C05496=1168.158,-99.130,-41.882,178.959,5.803,149.342
C05497=1168.163,-99.379,-41.873,178.956,5.803,149.343
C05498=1168.169,-99.629,-41.863,178.955,5.803,149.343
C05499=1168.174,-99.879,-41.854,178.952,5.803,149.344
C05500=1168.180,-100.128,-41.844,178.950,5.803,149.344
C05501=1168.185,-100.378,-41.835,178.948,5.802,149.345
C05502=1168.189,-100.629,-41.825,178.946,5.801,149.346
C05503=1168.195,-100.878,-41.815,178.944,5.802,149.346
C05504=1168.200,-101.128,-41.806,178.941,5.801,149.347
C05505=1168.206,-101.378,-41.796,178.940,5.801,149.347
C05506=1168.211,-101.628,-41.787,178.937,5.801,149.348
C05507=1168.216,-101.900,-41.777,178.935,5.800,149.349
C05508=1168.223,-102.171,-41.767,178.933,5.800,149.349
C05509=1168.229,-102.443,-41.756,178.930,5.800,149.350
C05510=1168.234,-102.715,-41.746,178.928,5.799,149.350
C05511=1168.239,-102.965,-41.737,178.926,5.799,149.351
C05512=1168.245,-103.214,-41.727,178.924,5.799,149.352
C05513=1168.250,-103.464,-41.718,178.922,5.799,149.352
C05514=1168.255,-103.714,-41.709,178.919,5.799,149.353
C05515=1168.261,-103.964,-41.699,178.917,5.798,149.353
C05516=1168.266,-104.213,-41.690,178.915,5.798,149.354
C05517=1168.271,-104.463,-41.681,178.913,5.797,149.355
C05518=1168.277,-104.713,-41.671,178.911,5.797,149.355
C05519=1168.282,-104.963,-41.662,178.909,5.797,149.356
C05520=1168.288,-105.213,-41.653,178.907,5.797,149.356
C05521=1168.293,-105.462,-41.643,178.905,5.796,149.357
C05522=1168.298,-105.712,-41.634,178.902,5.796,149.357
C05523=1168.304,-105.962,-41.625,178.900,5.796,149.358
C05524=1168.309,-106.211,-41.615,178.898,5.795,149.358
C05525=1168.314,-106.461,-41.606,178.896,5.796,149.359
C05526=1168.319,-106.711,-41.597,178.894,5.795,149.360
C05527=1168.325,-106.961,-41.588,178.892,5.795,149.360
C05528=1168.330,-107.210,-41.578,178.890,5.795,149.361
C05529=1168.335,-107.460,-41.569,178.888,5.795,149.361
C05530=1168.341,-107.710,-41.560,178.885,5.794,149.362
C05531=1168.346,-107.960,-41.551,178.883,5.793,149.362
C05532=1168.351,-108.209,-41.541,178.881,5.794,149.363
C05533=1168.357,-108.460,-41.532,178.879,5.793,149.364
C05534=1168.362,-108.709,-41.523,178.877,5.793,149.364
C05535=1168.367,-108.959,-41.514,178.875,5.793,149.365
C05536=1168.372,-109.209,-41.505,178.873,5.793,149.365
C05537=1168.378,-109.459,-41.495,178.871,5.792,149.366
C05538=1168.383,-109.709,-41.486,178.869,5.792,149.367
C05539=1168.388,-109.958,-41.477,178.867,5.792,149.367
C05540=1168.393,-110.208,-41.468,178.865,5.792,149.368
C05541=1168.400,-110.458,-41.459,178.862,5.791,149.368
C05542=1168.405,-110.707,-41.449,178.860,5.790,149.369
C05543=1168.410,-110.957,-41.440,178.858,5.791,149.369
C05544=1168.415,-111.207,-41.432,178.856,5.790,149.370
C05545=1168.421,-111.457,-41.422,178.854,5.790,149.370
C05546=1168.426,-111.707,-41.413,178.852,5.790,149.371
C05547=1168.431,-111.957,-41.404,178.850,5.790,149.372
C05548=1168.437,-112.206,-41.395,178.848,5.789,149.372
C05549=1168.442,-112.456,-41.386,178.846,5.789,149.373
C05550=1168.447,-112.706,-41.376,178.844,5.789,149.373
C05551=1168.452,-112.956,-41.367,178.842,5.789,149.374
C05552=1168.458,-113.206,-41.358,178.839,5.788,149.375
C05553=1168.463,-113.455,-41.350,178.838,5.788,149.375
C05554=1168.469,-113.704,-41.341,178.835,5.788,149.376
C05555=1168.474,-113.955,-41.331,178.833,5.787,149.376
C05556=1168.480,-114.205,-41.323,178.831,5.787,149.377
C05557=1168.485,-114.454,-41.314,178.829,5.787,149.377
C05558=1168.490,-114.704,-41.305,178.827,5.787,149.378
C05559=1168.495,-114.954,-41.296,178.825,5.786,149.378
C05560=1168.500,-115.204,-41.287,178.823,5.787,149.379
C05561=1168.507,-115.453,-41.278,178.820,5.786,149.380
C05562=1168.512,-115.703,-41.269,178.819,5.786,149.380
C05563=1168.517,-115.953,-41.260,178.816,5.785,149.381
C05564=1168.522,-116.203,-41.251,178.815,5.785,149.381
C05565=1168.528,-116.453,-41.242,178.812,5.785,149.382
C05566=1168.533,-116.703,-41.233,178.810,5.785,149.382
C05567=1168.538,-116.952,-41.224,178.808,5.784,149.383
C05568=1168.544,-117.202,-41.215,178.807,5.784,149.383
C05569=1168.550,-117.452,-41.206,178.804,5.784,149.384
C05570=1168.555,-117.702,-41.198,178.802,5.784,149.385
C05571=1168.560,-117.952,-41.189,178.800,5.783,149.385
C05572=1168.565,-118.201,-41.180,178.798,5.784,149.386
C05573=1168.570,-118.451,-41.171,178.796,5.783,149.386
C05574=1168.576,-118.700,-41.162,178.794,5.783,149.387
C05575=1168.581,-118.950,-41.153,178.792,5.783,149.388
C05576=1168.586,-119.200,-41.145,178.790,5.783,149.388
C05577=1168.591,-119.450,-41.136,178.788,5.782,149.389
C05578=1168.597,-119.700,-41.127,178.785,5.782,149.389
C05579=1168.603,-119.950,-41.117,178.783,5.782,149.390
C05580=1168.608,-120.199,-41.109,178.781,5.781,149.390
C05581=1168.613,-120.449,-41.100,178.779,5.781,149.391
C05582=1168.619,-120.699,-41.091,178.777,5.780,149.391
C05583=1168.624,-120.949,-41.082,178.775,5.780,149.392
C05584=1168.629,-121.198,-41.073,178.773,5.780,149.392
C05585=1168.635,-121.448,-41.065,178.771,5.780,149.393
C05586=1168.640,-121.698,-41.056,178.769,5.779,149.394
C05587=1168.645,-121.948,-41.048,178.767,5.779,149.394
C05588=1168.651,-122.198,-41.039,178.765,5.779,149.395
C05589=1168.656,-122.448,-41.030,178.763,5.779,149.395
C05590=1168.661,-122.697,-41.021,178.761,5.778,149.396
C05591=1168.667,-122.947,-41.012,178.759,5.779,149.396
C05592=1168.672,-123.197,-41.003,178.757,5.778,149.397
C05593=1168.677,-123.447,-40.995,178.755,5.778,149.397
C05594=1168.683,-123.696,-40.987,178.752,5.778,149.398
C05595=1168.688,-123.946,-40.978,178.751,5.778,149.399
C05596=1168.693,-124.196,-40.969,178.748,5.777,149.399
C05597=1168.699,-124.446,-40.960,178.747,5.777,149.400
C05598=1168.705,-124.695,-40.952,178.744,5.777,149.400
C05599=1168.710,-124.945,-40.943,178.743,5.777,149.401
C05600=1168.715,-125.195,-40.934,178.740,5.776,149.401
C05601=1168.720,-125.445,-40.925,178.738,5.776,149.402
C05602=1168.726,-125.694,-40.917,178.736,5.775,149.403
C05603=1168.731,-125.945,-40.909,178.735,5.776,149.403
C05604=1168.736,-126.194,-40.900,178.732,5.775,149.403
C05605=1168.742,-126.444,-40.891,178.730,5.775,149.404
C05606=1168.747,-126.693,-40.882,178.729,5.775,149.405
C05607=1168.753,-126.944,-40.874,178.726,5.774,149.405
C05608=1168.757,-127.193,-40.866,178.724,5.775,149.406
C05609=1168.762,-127.443,-40.857,178.722,5.774,149.406
C05610=1168.768,-127.692,-40.849,178.721,5.774,149.407
C05611=1168.347,-127.704,-40.890,178.717,5.777,149.409
C05612=1168.342,-127.455,-40.898,178.718,5.777,149.408
C05613=1168.337,-127.205,-40.907,178.720,5.778,149.408
C05614=1168.331,-126.954,-40.915,178.723,5.778,149.407
C05615=1168.326,-126.704,-40.924,178.725,5.778,149.407
C05616=1168.320,-126.455,-40.933,178.726,5.778,149.406
C05617=1168.315,-126.205,-40.942,178.729,5.779,149.405
C05618=1168.309,-125.955,-40.950,178.731,5.779,149.405
C05619=1168.304,-125.706,-40.958,178.733,5.780,149.404
C05620=1168.299,-125.456,-40.967,178.734,5.779,149.404
C05621=1168.294,-125.206,-40.976,178.737,5.780,149.403
C05622=1168.289,-124.956,-40.984,178.739,5.780,149.403
C05623=1168.283,-124.707,-40.992,178.741,5.781,149.402
C05624=1168.278,-124.457,-41.001,178.743,5.780,149.401
C05625=1168.273,-124.207,-41.010,178.745,5.781,149.401
C05626=1168.267,-123.957,-41.019,178.747,5.781,149.400
C05627=1168.262,-123.708,-41.027,178.749,5.782,149.400
C05628=1168.256,-123.458,-41.036,178.751,5.781,149.399
C05629=1168.251,-123.208,-41.045,178.753,5.782,149.399
C05630=1168.246,-122.958,-41.053,178.755,5.782,149.398
C05631=1168.241,-122.708,-41.062,178.758,5.782,149.398
C05632=1168.235,-122.459,-41.071,178.759,5.782,149.397
C05633=1168.230,-122.209,-41.080,178.761,5.783,149.397
C05634=1168.224,-121.959,-41.088,178.763,5.783,149.396
C05635=1168.219,-121.709,-41.097,178.766,5.783,149.395
C05636=1168.213,-121.460,-41.105,178.767,5.783,149.395
C05637=1168.208,-121.210,-41.114,178.769,5.784,149.394
C05638=1168.203,-120.960,-41.123,178.771,5.784,149.394
C05639=1168.197,-120.710,-41.133,178.774,5.784,149.393
C05640=1168.192,-120.460,-41.142,178.775,5.784,149.393
C05641=1168.186,-120.211,-41.150,178.778,5.785,149.392
C05642=1168.181,-119.961,-41.159,178.780,5.785,149.392
C05643=1168.176,-119.711,-41.168,178.782,5.786,149.391
C05644=1168.170,-119.460,-41.176,178.784,5.785,149.390
C05645=1168.165,-119.211,-41.185,178.786,5.786,149.390
C05646=1168.160,-118.961,-41.194,178.788,5.786,149.389
C05647=1168.154,-118.712,-41.202,178.790,5.786,149.389
C05648=1168.149,-118.462,-41.211,178.792,5.786,149.388
C05649=1168.144,-118.212,-41.220,178.794,5.787,149.388
C05650=1168.139,-117.962,-41.229,178.796,5.787,149.387
C05651=1168.134,-117.712,-41.238,178.798,5.787,149.386
C05652=1168.128,-117.462,-41.247,178.800,5.787,149.386
C05653=1168.122,-117.213,-41.256,178.803,5.788,149.385
C05654=1168.117,-116.963,-41.265,178.804,5.788,149.385
C05655=1168.112,-116.713,-41.274,178.806,5.788,149.384
C05656=1168.106,-116.463,-41.283,178.809,5.788,149.384
C05657=1168.101,-116.214,-41.292,178.811,5.789,149.383
C05658=1168.096,-115.964,-41.301,178.813,5.789,149.383
C05659=1168.090,-115.715,-41.309,178.815,5.789,149.382
C05660=1168.084,-115.464,-41.319,178.817,5.790,149.381
C05661=1168.079,-115.214,-41.327,178.819,5.790,149.381
C05662=1168.074,-114.965,-41.336,178.821,5.790,149.380
C05663=1168.069,-114.715,-41.345,178.823,5.790,149.380
C05664=1168.064,-114.465,-41.354,178.825,5.791,149.379
C05665=1168.059,-114.215,-41.363,178.827,5.790,149.379
C05666=1168.053,-113.965,-41.373,178.830,5.791,149.378
C05667=1168.047,-113.716,-41.382,178.831,5.791,149.378
C05668=1168.042,-113.467,-41.391,178.834,5.792,149.377
C05669=1168.037,-113.217,-41.400,178.835,5.792,149.376
C05670=1168.032,-112.967,-41.408,178.838,5.792,149.376
C05671=1168.027,-112.717,-41.417,178.840,5.792,149.375
C05672=1168.021,-112.467,-41.427,178.842,5.793,149.375
C05673=1168.015,-112.217,-41.436,178.843,5.793,149.374
C05674=1168.010,-111.967,-41.445,178.846,5.793,149.373
C05675=1168.005,-111.717,-41.454,178.848,5.794,149.373
C05676=1168.000,-111.468,-41.464,178.850,5.794,149.372
C05677=1167.994,-111.219,-41.472,178.853,5.794,149.372
C05678=1167.989,-110.969,-41.481,178.854,5.794,149.371
C05679=1167.983,-110.719,-41.490,178.857,5.794,149.371
C05680=1167.978,-110.469,-41.499,178.858,5.794,149.370
C05681=1167.972,-110.219,-41.508,178.861,5.795,149.370
C05682=1167.967,-109.969,-41.517,178.863,5.795,149.369
C05683=1167.962,-109.720,-41.527,178.865,5.796,149.368
C05684=1167.957,-109.470,-41.536,178.867,5.796,149.368
C05685=1167.951,-109.220,-41.545,178.869,5.796,149.367
C05686=1167.946,-108.970,-41.554,178.871,5.797,149.367
C05687=1167.941,-108.720,-41.563,178.873,5.797,149.366
C05688=1167.935,-108.471,-41.573,178.876,5.797,149.366
C05689=1167.930,-108.221,-41.582,178.877,5.797,149.365
C05690=1167.925,-107.971,-41.591,178.880,5.797,149.364
C05691=1167.920,-107.721,-41.600,178.882,5.797,149.364
C05692=1167.914,-107.471,-41.610,178.884,5.798,149.363
C05693=1167.909,-107.222,-41.619,178.886,5.798,149.363
C05694=1167.904,-106.972,-41.628,178.888,5.798,149.362
C05695=1167.898,-106.722,-41.638,178.890,5.799,149.362
C05696=1167.893,-106.472,-41.647,178.892,5.799,149.361
C05697=1167.888,-106.222,-41.656,178.895,5.800,149.360
C05698=1167.883,-105.973,-41.665,178.897,5.799,149.360
C05699=1167.877,-105.722,-41.674,178.899,5.800,149.359
C05700=1167.872,-105.473,-41.684,178.900,5.800,149.359
C05701=1167.867,-105.223,-41.693,178.903,5.800,149.358
C05702=1167.861,-104.973,-41.702,178.905,5.800,149.358
C05703=1167.856,-104.724,-41.712,178.907,5.801,149.357
C05704=1167.851,-104.474,-41.721,178.910,5.801,149.356
C05705=1167.845,-104.224,-41.730,178.911,5.801,149.356
C05706=1167.840,-103.975,-41.740,178.914,5.802,149.355
C05707=1167.834,-103.725,-41.750,178.915,5.802,149.355
C05708=1167.829,-103.475,-41.758,178.918,5.803,149.354
C05709=1167.824,-103.226,-41.768,178.920,5.802,149.354
C05710=1167.818,-102.975,-41.778,178.922,5.803,149.353
C05711=1167.813,-102.725,-41.786,178.925,5.803,149.352
C05712=1167.807,-102.454,-41.796,178.926,5.803,149.352
C05713=1167.802,-102.182,-41.807,178.929,5.804,149.351
C05714=1167.795,-101.910,-41.817,178.931,5.804,149.351
C05715=1167.790,-101.638,-41.828,178.933,5.804,149.350
C05716=1167.785,-101.389,-41.837,178.936,5.804,149.349
C05717=1167.779,-101.139,-41.847,178.938,5.805,149.349
C05718=1167.774,-100.889,-41.856,178.940,5.805,149.348
C05719=1167.769,-100.640,-41.865,178.942,5.805,149.348
C05720=1167.763,-100.390,-41.875,178.944,5.805,149.347
C05721=1167.758,-100.140,-41.884,178.947,5.806,149.346
C05722=1167.752,-99.890,-41.894,178.948,5.806,149.346
C05723=1167.748,-99.641,-41.903,178.950,5.807,149.345
C05724=1167.742,-99.391,-41.913,178.953,5.807,149.345
C05725=1167.736,-99.141,-41.922,178.955,5.807,149.344
C05726=1167.731,-98.891,-41.932,178.957,5.807,149.343
C05727=1167.726,-98.641,-41.941,178.959,5.807,149.343
C05728=1167.721,-98.391,-41.952,178.961,5.808,149.342
C05729=1167.716,-98.141,-41.960,178.964,5.808,149.342
C05730=1167.710,-97.892,-41.971,178.965,5.808,149.341
C05731=1167.705,-97.642,-41.980,178.968,5.809,149.341
C05732=1167.700,-97.393,-41.989,178.970,5.809,149.340
C05733=1167.694,-97.143,-41.999,178.972,5.810,149.340
C05734=1167.689,-96.893,-42.008,178.974,5.810,149.339
C05735=1167.683,-96.643,-42.018,178.976,5.810,149.338
C05736=1167.678,-96.394,-42.028,178.979,5.810,149.338
C05737=1167.673,-96.143,-42.037,178.980,5.810,149.337
C05738=1167.667,-95.894,-42.047,178.983,5.811,149.336
C05739=1167.663,-95.644,-42.057,178.985,5.811,149.336
C05740=1167.657,-95.394,-42.067,178.987,5.811,149.336
C05741=1167.652,-95.145,-42.076,178.989,5.812,149.335
C05742=1167.646,-94.895,-42.086,178.991,5.812,149.334
C05743=1167.641,-94.646,-42.095,178.994,5.812,149.334
C05744=1167.635,-94.395,-42.105,178.996,5.813,149.333
C05745=1167.631,-94.145,-42.115,178.998,5.813,149.332
C05746=1167.625,-93.896,-42.125,179.000,5.813,149.332
C05747=1167.620,-93.646,-42.134,179.002,5.813,149.331
C05748=1167.615,-93.397,-42.144,179.004,5.814,149.331
C05749=1167.609,-93.146,-42.154,179.007,5.815,149.330
C05750=1167.604,-92.897,-42.163,179.009,5.814,149.330
C05751=1167.599,-92.647,-42.174,179.011,5.815,149.329
C05752=1167.594,-92.397,-42.183,179.013,5.814,149.328
C05753=1167.588,-92.148,-42.193,179.015,5.815,149.328
C05754=1167.583,-91.898,-42.202,179.018,5.816,149.327
C05755=1167.577,-91.648,-42.212,179.019,5.816,149.327
C05756=1167.572,-91.399,-42.222,179.022,5.816,149.326
C05757=1167.567,-91.149,-42.232,179.024,5.816,149.325
C05758=1167.561,-90.898,-42.242,179.026,5.817,149.325
C05759=1167.556,-90.649,-42.252,179.029,5.817,149.324
C05760=1167.551,-90.400,-42.261,179.030,5.817,149.324
C05761=1167.545,-90.150,-42.271,179.033,5.818,149.323
C05762=1167.541,-89.900,-42.281,179.035,5.818,149.323
C05763=1167.535,-89.650,-42.291,179.037,5.818,149.322
C05764=1167.529,-89.400,-42.301,179.039,5.819,149.321
C05765=1167.525,-89.151,-42.310,179.041,5.819,149.321
C05766=1167.519,-88.901,-42.320,179.044,5.819,149.320
C05767=1167.514,-88.651,-42.331,179.046,5.820,149.320
C05768=1167.509,-88.401,-42.340,179.048,5.819,149.319
C05769=1167.503,-88.151,-42.350,179.050,5.820,149.319
C05770=1167.498,-87.902,-42.360,179.053,5.821,149.318
C05771=1167.493,-87.653,-42.370,179.054,5.821,149.317
C05772=1167.487,-87.402,-42.380,179.057,5.821,149.317
C05773=1167.482,-87.152,-42.390,179.059,5.821,149.316
C05774=1167.477,-86.903,-42.400,179.061,5.821,149.315
C05775=1167.471,-86.654,-42.410,179.063,5.822,149.315
C05776=1167.466,-86.403,-42.420,179.065,5.822,149.314
C05777=1167.461,-86.153,-42.429,179.068,5.822,149.314
C05778=1167.456,-85.904,-42.440,179.070,5.823,149.313
C05779=1167.450,-85.654,-42.450,179.072,5.823,149.313
C05780=1167.445,-85.404,-42.460,179.074,5.824,149.312
C05781=1167.440,-85.155,-42.470,179.077,5.824,149.311
C05782=1167.435,-84.905,-42.480,179.078,5.824,149.311
C05783=1167.429,-84.654,-42.490,179.081,5.824,149.310
C05784=1167.424,-84.405,-42.500,179.083,5.825,149.310
C05785=1167.419,-84.156,-42.510,179.085,5.825,149.309
C05786=1167.413,-83.906,-42.520,179.088,5.826,149.309
C05787=1167.408,-83.656,-42.531,179.090,5.825,149.308
C05788=1167.403,-83.407,-42.540,179.092,5.826,149.307
C05789=1167.398,-83.157,-42.550,179.094,5.827,149.307
C05790=1167.393,-82.907,-42.561,179.096,5.826,149.306
C05791=1167.387,-82.657,-42.571,179.098,5.827,149.306
C05792=1167.382,-82.407,-42.580,179.101,5.827,149.305
C05793=1167.376,-82.158,-42.590,179.103,5.827,149.304
C05794=1167.371,-81.908,-42.601,179.105,5.828,149.304
C05795=1167.366,-81.658,-42.611,179.107,5.829,149.303
C05796=1167.360,-81.409,-42.621,179.110,5.828,149.303
C05797=1167.356,-81.159,-42.631,179.112,5.829,149.302
C05798=1167.350,-80.909,-42.641,179.114,5.829,149.301
C05799=1167.345,-80.660,-42.652,179.116,5.829,149.301
C05800=1167.340,-80.409,-42.662,179.119,5.830,149.300
C05801=1167.334,-80.160,-42.672,179.121,5.831,149.300
C05802=1167.328,-79.910,-42.683,179.123,5.830,149.299
C05803=1167.324,-79.660,-42.693,179.125,5.831,149.299
C05804=1167.319,-79.411,-42.703,179.128,5.831,149.298
C05805=1167.313,-79.161,-42.713,179.129,5.831,149.297
C05806=1167.308,-78.911,-42.724,179.132,5.832,149.297
C05807=1167.302,-78.661,-42.734,179.134,5.833,149.296
C05808=1167.297,-78.412,-42.744,179.136,5.832,149.295
C05809=1167.292,-78.162,-42.755,179.138,5.833,149.295
C05810=1167.287,-77.912,-42.764,179.141,5.833,149.294
C05811=1167.281,-77.663,-42.774,179.143,5.833,149.294
C05812=1167.276,-77.413,-42.785,179.145,5.834,149.293
C05813=1167.271,-77.163,-42.795,179.148,5.834,149.293
C05814=1167.265,-76.914,-42.805,179.150,5.834,149.292
C05815=1167.260,-76.663,-42.816,179.152,5.835,149.291
C05816=1167.254,-76.393,-42.827,179.155,5.835,149.291
C05817=1167.249,-76.122,-42.839,179.157,5.836,149.290
C05818=1167.243,-75.850,-42.850,179.159,5.836,149.289
C05819=1167.237,-75.580,-42.861,179.162,5.836,149.289
C05820=1167.232,-75.329,-42.872,179.164,5.837,149.288
C05821=1167.226,-75.080,-42.882,179.166,5.837,149.288
C05822=1167.221,-74.829,-42.892,179.168,5.837,149.287
C05823=1167.216,-74.580,-42.903,179.171,5.838,149.286
C05824=1167.211,-74.331,-42.913,179.173,5.838,149.286
C05825=1167.206,-74.081,-42.924,179.175,5.838,149.285
C05826=1167.200,-73.831,-42.934,179.177,5.839,149.285
C05827=1167.195,-73.581,-42.945,179.180,5.839,149.284
C05828=1167.189,-73.331,-42.955,179.182,5.840,149.284
C05829=1167.184,-73.081,-42.966,179.184,5.840,149.283
C05830=1167.179,-72.832,-42.976,179.186,5.840,149.282
C05831=1167.174,-72.583,-42.987,179.189,5.841,149.282
C05832=1167.169,-72.332,-42.997,179.190,5.841,149.281
C05833=1167.163,-72.083,-43.007,179.193,5.841,149.280
C05834=1167.158,-71.833,-43.018,179.195,5.842,149.280
C05835=1167.152,-71.583,-43.028,179.197,5.842,149.279
C05836=1167.148,-71.334,-43.040,179.200,5.842,149.279
C05837=1167.142,-71.084,-43.050,179.202,5.843,149.278
C05838=1167.136,-70.834,-43.060,179.204,5.844,149.278
C05839=1167.131,-70.584,-43.071,179.207,5.843,149.277
C05840=1167.126,-70.335,-43.081,179.209,5.844,149.276
C05841=1167.121,-70.085,-43.092,179.211,5.844,149.276
C05842=1167.116,-69.835,-43.102,179.213,5.844,149.275
C05843=1167.111,-69.585,-43.113,179.216,5.845,149.274
C05844=1167.105,-69.336,-43.124,179.218,5.845,149.274
C05845=1167.100,-69.086,-43.134,179.220,5.845,149.273
C05846=1167.095,-68.837,-43.145,179.222,5.846,149.273
C05847=1167.090,-68.587,-43.156,179.225,5.846,149.272
C05848=1167.084,-68.337,-43.166,179.227,5.847,149.271
C05849=1167.079,-68.087,-43.177,179.229,5.847,149.271
C05850=1167.074,-67.838,-43.188,179.232,5.847,149.270
C05851=1167.069,-67.588,-43.198,179.234,5.848,149.270
C05852=1167.063,-67.338,-43.209,179.236,5.847,149.269
C05853=1167.058,-67.088,-43.220,179.238,5.848,149.269
C05854=1167.052,-66.839,-43.230,179.241,5.849,149.268
C05855=1167.047,-66.589,-43.241,179.243,5.849,149.267
C05856=1167.042,-66.340,-43.252,179.245,5.849,149.267
C05857=1167.037,-66.090,-43.263,179.247,5.850,149.266
C05858=1167.032,-65.840,-43.273,179.250,5.850,149.265
C05859=1167.027,-65.590,-43.284,179.252,5.851,149.265
C05860=1167.021,-65.341,-43.294,179.254,5.851,149.264
C05861=1167.016,-65.091,-43.306,179.256,5.851,149.264
C05862=1167.010,-64.841,-43.316,179.259,5.852,149.263
C05863=1167.005,-64.591,-43.327,179.261,5.852,149.263
C05864=1167.001,-64.341,-43.338,179.263,5.852,149.262
C05865=1166.995,-64.092,-43.348,179.266,5.853,149.261
C05866=1166.990,-63.842,-43.360,179.268,5.853,149.261
C05867=1166.985,-63.593,-43.370,179.270,5.853,149.260
C05868=1166.979,-63.343,-43.382,179.272,5.854,149.260
C05869=1166.974,-63.093,-43.392,179.275,5.855,149.259
C05870=1166.969,-62.844,-43.403,179.277,5.855,149.258
C05871=1166.963,-62.594,-43.413,179.279,5.855,149.258
C05872=1166.958,-62.344,-43.424,179.282,5.855,149.257
C05873=1166.953,-62.094,-43.436,179.284,5.856,149.256
C05874=1166.947,-61.844,-43.446,179.286,5.857,149.256
C05875=1166.943,-61.595,-43.457,179.289,5.856,149.255
C05876=1166.937,-61.345,-43.468,179.291,5.857,149.255
C05877=1166.932,-61.096,-43.479,179.293,5.857,149.254
C05878=1166.927,-60.846,-43.491,179.296,5.858,149.254
C05879=1166.921,-60.596,-43.501,179.298,5.858,149.253
C05880=1166.917,-60.346,-43.512,179.300,5.859,149.252
C05881=1166.911,-60.097,-43.523,179.302,5.859,149.252
C05882=1166.906,-59.847,-43.534,179.305,5.860,149.251
C05883=1166.901,-59.597,-43.545,179.307,5.859,149.251
C05884=1166.895,-59.348,-43.556,179.309,5.860,149.250
C05885=1166.890,-59.098,-43.566,179.312,5.861,149.249
C05886=1166.886,-58.848,-43.578,179.314,5.861,149.249
C05887=1166.880,-58.599,-43.589,179.316,5.861,149.248
C05888=1166.875,-58.348,-43.600,179.319,5.861,149.247
C05889=1166.869,-58.100,-43.611,179.321,5.862,149.247
C05890=1166.864,-57.849,-43.622,179.323,5.863,149.246
C05891=1166.859,-57.599,-43.633,179.325,5.863,149.246
C05892=1166.854,-57.350,-43.644,179.328,5.863,149.245
C05893=1166.849,-57.100,-43.655,179.330,5.864,149.245
C05894=1166.843,-56.850,-43.667,179.332,5.864,149.244
C05895=1166.838,-56.601,-43.678,179.334,5.864,149.243
C05896=1166.833,-56.351,-43.688,179.337,5.865,149.243
C05897=1166.827,-56.101,-43.700,179.339,5.865,149.242
C05898=1166.822,-55.852,-43.711,179.342,5.866,149.242
C05899=1166.817,-55.602,-43.722,179.344,5.866,149.241
C05900=1166.812,-55.352,-43.733,179.346,5.866,149.240
C05901=1166.806,-55.103,-43.744,179.349,5.867,149.240
C05902=1166.801,-54.853,-43.755,179.351,5.868,149.239
C05903=1166.796,-54.603,-43.767,179.353,5.868,149.239
C05904=1166.791,-54.354,-43.778,179.355,5.868,149.238
C05905=1166.786,-54.104,-43.789,179.358,5.868,149.237
C05906=1166.780,-53.854,-43.800,179.360,5.869,149.237
C05907=1166.776,-53.604,-43.811,179.363,5.870,149.236
C05908=1166.770,-53.355,-43.822,179.365,5.870,149.235
C05909=1166.765,-53.105,-43.834,179.367,5.870,149.235
C05910=1166.760,-52.855,-43.845,179.369,5.870,149.234
C05911=1166.754,-52.606,-43.856,179.372,5.871,149.234
C05912=1166.749,-52.356,-43.868,179.374,5.872,149.233
C05913=1166.744,-52.107,-43.879,179.376,5.872,149.233
C05914=1166.739,-51.856,-43.890,179.379,5.872,149.232
C05915=1166.733,-51.607,-43.901,179.381,5.873,149.231
C05916=1166.728,-51.357,-43.913,179.383,5.873,149.231
C05917=1166.723,-51.108,-43.924,179.386,5.874,149.230
C05918=1166.719,-50.858,-43.935,179.388,5.874,149.230
C05919=1166.712,-50.608,-43.946,179.390,5.874,149.229
C05920=1166.707,-50.338,-43.959,179.392,5.875,149.228
C05921=1166.701,-50.067,-43.972,179.395,5.875,149.228
C05922=1166.695,-49.797,-43.984,179.398,5.876,149.227
C05923=1166.691,-49.526,-43.996,179.401,5.876,149.226
C05924=1166.685,-49.277,-44.008,179.403,5.877,149.226
C05925=1166.680,-49.028,-44.019,179.405,5.877,149.225
C05926=1166.674,-48.777,-44.030,179.407,5.877,149.225
C05927=1166.669,-48.527,-44.041,179.410,5.878,149.224
C05928=1166.664,-48.277,-44.053,179.412,5.878,149.223
C05929=1166.659,-48.029,-44.064,179.414,5.879,149.223
C05930=1166.653,-47.779,-44.076,179.417,5.879,149.222
C05931=1166.649,-47.529,-44.087,179.419,5.880,149.222
C05932=1166.643,-47.279,-44.099,179.421,5.880,149.221
C05933=1166.638,-47.029,-44.110,179.424,5.881,149.220
C05934=1166.632,-46.780,-44.122,179.426,5.881,149.220
C05935=1166.627,-46.530,-44.134,179.428,5.882,149.219
C05936=1166.622,-46.281,-44.145,179.431,5.882,149.218
C05937=1166.617,-46.031,-44.157,179.433,5.882,149.218
C05938=1166.612,-45.781,-44.168,179.435,5.883,149.217
C05939=1166.606,-45.532,-44.180,179.438,5.883,149.217
C05940=1166.601,-45.282,-44.191,179.440,5.884,149.216
C05941=1166.596,-45.032,-44.203,179.443,5.884,149.215
C05942=1166.591,-44.783,-44.214,179.445,5.885,149.215
C05943=1166.586,-44.533,-44.226,179.447,5.885,149.214
C05944=1166.581,-44.284,-44.237,179.450,5.885,149.214
C05945=1166.575,-44.034,-44.249,179.452,5.886,149.213
C05946=1166.570,-43.784,-44.261,179.455,5.886,149.212
C05947=1166.565,-43.534,-44.272,179.457,5.887,149.212
C05948=1166.560,-43.284,-44.284,179.459,5.887,149.211
C05949=1166.555,-43.035,-44.295,179.461,5.888,149.211
C05950=1166.550,-42.785,-44.307,179.464,5.888,149.210
C05951=1166.543,-42.536,-44.319,179.466,5.889,149.210
C05952=1166.539,-42.286,-44.330,179.469,5.889,149.209
C05953=1166.533,-42.036,-44.342,179.471,5.890,149.208
C05954=1166.528,-41.786,-44.354,179.473,5.890,149.208
C05955=1166.523,-41.536,-44.365,179.475,5.890,149.207
C05956=1166.518,-41.286,-44.377,179.478,5.891,149.206
C05957=1166.513,-41.037,-44.389,179.480,5.891,149.206
C05958=1166.508,-40.788,-44.401,179.483,5.892,149.205
C05959=1166.502,-40.538,-44.412,179.485,5.893,149.205
C05960=1166.497,-40.289,-44.423,179.488,5.893,149.204
C05961=1166.492,-40.039,-44.435,179.489,5.893,149.203
C05962=1166.486,-39.789,-44.447,179.492,5.893,149.203
C05963=1166.482,-39.539,-44.458,179.494,5.894,149.202
C05964=1166.477,-39.290,-44.471,179.497,5.895,149.202
C05965=1166.471,-39.040,-44.483,179.499,5.895,149.201
C05966=1166.466,-38.790,-44.495,179.502,5.896,149.200
C05967=1166.461,-38.540,-44.506,179.504,5.896,149.200
C05968=1166.456,-38.290,-44.518,179.506,5.896,149.199
C05969=1166.450,-38.042,-44.530,179.509,5.897,149.199
C05970=1166.445,-37.792,-44.542,179.511,5.897,149.198
C05971=1166.440,-37.542,-44.553,179.514,5.898,149.197
C05972=1166.434,-37.292,-44.565,179.516,5.899,149.197
C05973=1166.429,-37.042,-44.577,179.518,5.899,149.196
C05974=1166.425,-36.793,-44.589,179.521,5.900,149.195
C05975=1166.419,-36.543,-44.601,179.523,5.900,149.195
C05976=1166.414,-36.293,-44.613,179.525,5.900,149.194
C05977=1166.408,-36.044,-44.625,179.528,5.901,149.194
C05978=1166.404,-35.795,-44.637,179.530,5.901,149.193
C05979=1166.398,-35.545,-44.649,179.533,5.902,149.192
C05980=1166.393,-35.295,-44.661,179.535,5.902,149.192
C05981=1166.388,-35.045,-44.673,179.538,5.903,149.191
C05982=1166.383,-34.796,-44.685,179.540,5.904,149.191
C05983=1166.378,-34.546,-44.696,179.542,5.903,149.190
C05984=1166.373,-34.296,-44.709,179.544,5.904,149.190
C05985=1166.367,-34.047,-44.721,179.547,5.905,149.189
C05986=1166.362,-33.797,-44.733,179.549,5.905,149.188
C05987=1166.357,-33.548,-44.745,179.552,5.906,149.188
C05988=1166.352,-33.298,-44.757,179.554,5.906,149.187
C05989=1166.347,-33.048,-44.769,179.556,5.907,149.187
C05990=1166.341,-32.798,-44.781,179.559,5.907,149.186
C05991=1166.336,-32.548,-44.793,179.561,5.907,149.185
C05992=1166.331,-32.299,-44.805,179.563,5.908,149.185
C05993=1166.326,-32.050,-44.817,179.566,5.908,149.184
C05994=1166.321,-31.800,-44.829,179.568,5.909,149.184
C05995=1166.316,-31.550,-44.841,179.571,5.910,149.183
C05996=1166.310,-31.300,-44.853,179.573,5.910,149.182
C05997=1166.305,-31.051,-44.866,179.576,5.911,149.182
C05998=1166.300,-30.801,-44.878,179.578,5.911,149.181
C05999=1166.294,-30.551,-44.890,179.581,5.912,149.180
C06000=1166.289,-30.302,-44.902,179.583,5.912,149.180
C06001=1166.284,-30.052,-44.914,179.585,5.913,149.179
C06002=1166.279,-29.803,-44.926,179.587,5.913,149.179
C06003=1166.274,-29.553,-44.938,179.590,5.914,149.178
C06004=1166.269,-29.304,-44.951,179.592,5.914,149.177
C06005=1166.263,-29.054,-44.963,179.595,5.915,149.177
C06006=1166.258,-28.804,-44.975,179.597,5.915,149.176
C06007=1166.253,-28.554,-44.987,179.600,5.916,149.176
C06008=1166.248,-28.305,-45.000,179.602,5.917,149.175
C06009=1166.243,-28.054,-45.012,179.605,5.917,149.174
C06010=1166.238,-27.805,-45.025,179.607,5.918,149.174
C06011=1166.232,-27.555,-45.036,179.609,5.918,149.173
C06012=1166.227,-27.306,-45.049,179.612,5.918,149.173
C06013=1166.222,-27.056,-45.060,179.614,5.919,149.172
C06014=1166.217,-26.807,-45.073,179.616,5.919,149.171
C06015=1166.212,-26.558,-45.085,179.619,5.920,149.171
C06016=1166.207,-26.308,-45.097,179.621,5.920,149.170
C06017=1166.202,-26.058,-45.110,179.624,5.921,149.170
C06018=1166.196,-25.808,-45.122,179.626,5.922,149.169
C06019=1166.191,-25.559,-45.134,179.629,5.922,149.168
C06020=1166.186,-25.309,-45.147,179.631,5.923,149.168
C06021=1166.181,-25.059,-45.159,179.634,5.923,149.167
C06022=1166.176,-24.810,-45.172,179.636,5.924,149.167
C06023=1166.171,-24.560,-45.184,179.638,5.925,149.166
C06024=1166.165,-24.290,-45.198,179.641,5.925,149.165
C06025=1166.159,-24.020,-45.211,179.644,5.926,149.165
C06026=1166.154,-23.751,-45.224,179.646,5.926,149.164
C06027=1166.148,-23.480,-45.239,179.649,5.927,149.163
C06028=1166.143,-23.231,-45.251,179.651,5.927,149.163
C06029=1166.138,-22.981,-45.263,179.653,5.928,149.162
C06030=1166.132,-22.732,-45.276,179.656,5.928,149.162
C06031=1166.127,-22.482,-45.288,179.659,5.929,149.161
C06032=1166.122,-22.233,-45.300,179.661,5.930,149.160
C06033=1166.117,-21.983,-45.313,179.663,5.929,149.160
C06034=1166.112,-21.733,-45.325,179.665,5.930,149.159
C06035=1166.107,-21.483,-45.338,179.668,5.931,149.159
C06036=1166.102,-21.234,-45.350,179.671,5.931,149.158
C06037=1166.097,-20.985,-45.363,179.673,5.932,149.157
C06038=1166.091,-20.735,-45.375,179.675,5.932,149.157
C06039=1166.087,-20.485,-45.388,179.678,5.933,149.156
C06040=1166.081,-20.235,-45.401,179.680,5.934,149.156
C06041=1166.076,-19.986,-45.413,179.682,5.934,149.155
C06042=1166.070,-19.736,-45.425,179.685,5.935,149.154
C06043=1166.065,-19.487,-45.438,179.688,5.935,149.154
C06044=1166.061,-19.237,-45.451,179.690,5.936,149.153
C06045=1166.055,-18.987,-45.464,179.693,5.936,149.153
C06046=1166.050,-18.738,-45.476,179.695,5.937,149.152
C06047=1166.044,-18.488,-45.489,179.697,5.938,149.151
C06048=1166.039,-18.238,-45.501,179.700,5.938,149.151
C06049=1166.034,-17.988,-45.514,179.702,5.939,149.150
C06050=1166.029,-17.739,-45.527,179.705,5.939,149.150
C06051=1166.024,-17.490,-45.539,179.707,5.940,149.149
C06052=1166.019,-17.240,-45.552,179.710,5.941,149.148
C06053=1166.014,-16.990,-45.566,179.712,5.941,149.148
C06054=1166.008,-16.740,-45.577,179.715,5.942,149.147
C06055=1166.003,-16.491,-45.590,179.717,5.942,149.146
C06056=1165.998,-16.241,-45.603,179.719,5.943,149.146
C06057=1165.994,-15.991,-45.616,179.722,5.944,149.145
C06058=1165.988,-15.742,-45.629,179.724,5.944,149.145
C06059=1165.983,-15.493,-45.641,179.726,5.944,149.144
C06060=1165.978,-15.243,-45.654,179.729,5.945,149.143
C06061=1165.973,-14.993,-45.667,179.731,5.945,149.143
C06062=1165.968,-14.744,-45.680,179.734,5.946,149.142
C06063=1165.962,-14.494,-45.693,179.736,5.947,149.142
C06064=1165.957,-14.245,-45.705,179.739,5.947,149.141
C06065=1165.952,-13.995,-45.718,179.741,5.948,149.140
C06066=1165.947,-13.746,-45.731,179.743,5.948,149.140
C06067=1165.941,-13.496,-45.744,179.746,5.949,149.139
C06068=1165.937,-13.246,-45.757,179.748,5.950,149.139
C06069=1165.932,-12.997,-45.770,179.751,5.950,149.138
C06070=1165.926,-12.747,-45.783,179.754,5.950,149.137
C06071=1165.921,-12.497,-45.796,179.756,5.951,149.137
C06072=1165.916,-12.248,-45.808,179.758,5.952,149.136
C06073=1165.911,-11.998,-45.821,179.761,5.953,149.136
C06074=1165.906,-11.748,-45.835,179.763,5.953,149.135
C06075=1165.901,-11.499,-45.847,179.765,5.954,149.135
C06076=1165.896,-11.249,-45.860,179.768,5.954,149.134
C06077=1165.890,-10.999,-45.873,179.771,5.955,149.133
C06078=1165.885,-10.750,-45.886,179.773,5.956,149.133
C06079=1165.880,-10.500,-45.899,179.776,5.956,149.132
C06080=1165.875,-10.250,-45.912,179.778,5.957,149.132
C06081=1165.870,-10.001,-45.925,179.780,5.957,149.131
C06082=1165.865,-9.751,-45.937,179.783,5.958,149.130
C06083=1165.860,-9.502,-45.952,179.785,5.959,149.130
C06084=1165.855,-9.252,-45.964,179.788,5.959,149.129
C06085=1165.849,-9.003,-45.977,179.790,5.960,149.129
C06086=1165.844,-8.753,-45.990,179.793,5.960,149.128
C06087=1165.839,-8.503,-46.003,179.795,5.961,149.127
C06088=1165.833,-8.254,-46.016,179.798,5.962,149.127
C06089=1165.829,-8.004,-46.029,179.800,5.962,149.126
C06090=1165.824,-7.755,-46.042,179.802,5.963,149.126
C06091=1165.819,-7.505,-46.056,179.805,5.963,149.125
C06092=1165.813,-7.255,-46.069,179.807,5.964,149.124
C06093=1165.808,-7.006,-46.081,179.810,5.965,149.124
C06094=1165.803,-6.756,-46.095,179.813,5.965,149.123
C06095=1165.798,-6.507,-46.108,179.815,5.967,149.123
C06096=1165.793,-6.257,-46.122,179.818,5.967,149.122
C06097=1165.788,-6.007,-46.134,179.820,5.968,149.121
C06098=1165.782,-5.758,-46.147,179.823,5.968,149.121
C06099=1165.778,-5.508,-46.161,179.825,5.969,149.120
C06100=1165.772,-5.259,-46.174,179.828,5.970,149.120
C06101=1165.767,-5.009,-46.187,179.830,5.970,149.119
C06102=1165.762,-4.759,-46.200,179.832,5.971,149.118
C06103=1165.757,-4.510,-46.214,179.835,5.971,149.118
C06104=1165.752,-4.260,-46.227,179.837,5.972,149.117
C06105=1165.747,-4.010,-46.240,179.840,5.973,149.117
C06106=1165.742,-3.761,-46.253,179.843,5.973,149.116
C06107=1165.736,-3.512,-46.267,179.845,5.974,149.115
C06108=1165.732,-3.262,-46.280,179.847,5.974,149.115
C06109=1165.726,-3.012,-46.293,179.850,5.975,149.114
C06110=1165.722,-2.763,-46.307,179.852,5.976,149.114
C06111=1165.716,-2.513,-46.320,179.855,5.976,149.113
C06112=1165.711,-2.263,-46.333,179.857,5.977,149.112
C06113=1165.706,-2.014,-46.347,179.860,5.977,149.112
C06114=1165.700,-1.764,-46.360,179.862,5.978,149.111
C06115=1165.696,-1.515,-46.374,179.865,5.979,149.111
C06116=1165.690,-1.265,-46.387,179.867,5.979,149.110
C06117=1165.685,-1.015,-46.400,179.869,5.980,149.109
C06118=1165.680,-0.766,-46.414,179.873,5.981,149.109
C06119=1165.675,-0.516,-46.427,179.875,5.982,149.108
C06120=1165.670,-0.267,-46.441,179.877,5.982,149.108
C06121=1165.664,-0.017,-46.454,179.880,5.983,149.107
C06122=1165.660,0.233,-46.467,179.882,5.984,149.106
C06123=1165.654,0.482,-46.481,179.885,5.984,149.106
C06124=1165.650,0.732,-46.494,179.887,5.985,149.105
C06125=1165.644,0.981,-46.508,179.890,5.985,149.105
C06126=1165.640,1.231,-46.521,179.892,5.986,149.104
C06127=1165.634,1.480,-46.535,179.895,5.987,149.104
C06128=1165.629,1.749,-46.550,179.897,5.987,149.103
C06129=1165.623,2.019,-46.564,179.900,5.989,149.102
C06130=1165.618,2.288,-46.578,179.903,5.989,149.102
C06131=1165.612,2.557,-46.593,179.905,5.990,149.101
C06132=1165.607,2.808,-46.607,179.908,5.990,149.100
C06133=1165.601,3.057,-46.621,179.910,5.991,149.100
C06134=1165.597,3.307,-46.634,179.913,5.991,149.099
C06135=1165.591,3.556,-46.647,179.915,5.992,149.099
C06136=1165.586,3.805,-46.662,179.918,5.993,149.098
C06137=1165.582,4.055,-46.675,179.921,5.994,149.097
C06138=1165.576,4.304,-46.689,179.923,5.995,149.097
C06139=1165.571,4.555,-46.702,179.926,5.995,149.096
C06140=1165.566,4.803,-46.715,179.928,5.996,149.096
C06141=1165.561,5.054,-46.729,179.931,5.997,149.095
C06142=1165.555,5.303,-46.743,179.933,5.997,149.095
C06143=1165.551,5.552,-46.757,179.935,5.998,149.094
C06144=1165.546,5.803,-46.770,179.938,5.998,149.093
C06145=1165.540,6.052,-46.784,179.940,5.999,149.093
C06146=1165.535,6.301,-46.798,179.943,6.000,149.092
C06147=1165.530,6.551,-46.811,179.945,6.000,149.092
C06148=1165.525,6.800,-46.825,179.948,6.002,149.091
C06149=1165.520,7.050,-46.840,179.951,6.002,149.090
C06150=1165.515,7.300,-46.853,179.953,6.003,149.090
C06151=1165.510,7.549,-46.866,179.956,6.003,149.089
C06152=1165.505,7.799,-46.881,179.958,6.004,149.089
C06153=1165.499,8.048,-46.894,179.961,6.005,149.088
C06154=1165.495,8.298,-46.908,179.963,6.006,149.087
C06155=1165.490,8.547,-46.922,179.965,6.006,149.087
C06156=1165.485,8.796,-46.936,179.968,6.007,149.086
C06157=1165.479,9.047,-46.949,179.971,6.008,149.086
C06158=1165.474,9.296,-46.963,179.973,6.009,149.085
C06159=1165.469,9.546,-46.978,179.976,6.009,149.084
C06160=1165.465,9.795,-46.991,179.978,6.010,149.084
C06161=1165.459,10.045,-47.004,179.980,6.011,149.083
C06162=1165.454,10.294,-47.019,179.983,6.011,149.083
C06163=1165.449,10.544,-47.033,179.986,6.012,149.082
C06164=1165.443,10.793,-47.047,179.988,6.013,149.081
C06165=1165.438,11.043,-47.060,179.991,6.014,149.081
C06166=1165.434,11.293,-47.074,179.993,6.015,149.080
C06167=1165.429,11.542,-47.088,179.996,6.015,149.080
C06168=1165.423,11.791,-47.102,179.998,6.016,149.079
C06169=1165.418,12.041,-47.117,-179.999,6.016,149.079
C06170=1165.414,12.291,-47.131,-179.997,6.017,149.078
C06171=1165.408,12.540,-47.144,-179.994,6.018,149.077
C06172=1165.403,12.790,-47.158,-179.992,6.018,149.077
C06173=1165.398,13.040,-47.173,-179.989,6.020,149.076
C06174=1165.393,13.289,-47.186,-179.986,6.020,149.076
C06175=1165.388,13.538,-47.200,-179.984,6.021,149.075
C06176=1165.383,13.788,-47.214,-179.982,6.022,149.074
C06177=1165.378,14.038,-47.229,-179.979,6.022,149.074
C06178=1165.373,14.287,-47.243,-179.977,6.023,149.073
C06179=1165.368,14.536,-47.257,-179.974,6.023,149.073
C06180=1165.363,14.786,-47.271,-179.971,6.025,149.072
C06181=1165.357,15.036,-47.285,-179.969,6.025,149.071
C06182=1165.352,15.285,-47.299,-179.966,6.026,149.071
C06183=1165.347,15.535,-47.313,-179.964,6.027,149.070
C06184=1165.342,15.785,-47.327,-179.961,6.027,149.070
C06185=1165.337,16.035,-47.342,-179.959,6.028,149.069
C06186=1165.331,16.284,-47.355,-179.956,6.029,149.068
C06187=1165.326,16.533,-47.370,-179.954,6.030,149.068
C06188=1165.321,16.783,-47.384,-179.951,6.031,149.067
C06189=1165.317,17.033,-47.398,-179.949,6.031,149.067
C06190=1165.312,17.282,-47.413,-179.946,6.032,149.066
C06191=1165.306,17.531,-47.426,-179.943,6.032,149.066
C06192=1165.301,17.781,-47.441,-179.941,6.034,149.065
C06193=1165.296,18.031,-47.455,-179.938,6.035,149.064
C06194=1165.291,18.280,-47.470,-179.936,6.035,149.064
C06195=1165.286,18.530,-47.484,-179.933,6.036,149.063
C06196=1165.281,18.779,-47.498,-179.931,6.037,149.063
C06197=1165.276,19.028,-47.512,-179.928,6.037,149.062
C06198=1165.271,19.278,-47.527,-179.926,6.039,149.062
C06199=1165.266,19.528,-47.541,-179.923,6.039,149.061
C06200=1165.261,19.778,-47.555,-179.920,6.040,149.060
C06201=1165.256,20.027,-47.569,-179.918,6.041,149.060
C06202=1165.251,20.276,-47.583,-179.916,6.041,149.059
C06203=1165.246,20.526,-47.598,-179.913,6.042,149.059
C06204=1165.241,20.775,-47.613,-179.910,6.043,149.058
C06205=1165.236,21.025,-47.627,-179.908,6.044,149.058
C06206=1165.231,21.274,-47.641,-179.905,6.044,149.057
C06207=1165.226,21.523,-47.655,-179.903,6.045,149.056
C06208=1165.220,21.774,-47.670,-179.901,6.046,149.056
C06209=1165.215,22.023,-47.684,-179.897,6.047,149.055
C06210=1165.210,22.272,-47.699,-179.895,6.048,149.055
C06211=1165.205,22.522,-47.714,-179.892,6.048,149.054
C06212=1165.200,22.772,-47.728,-179.890,6.049,149.053
C06213=1165.195,23.021,-47.742,-179.888,6.050,149.053
C06214=1165.190,23.271,-47.756,-179.885,6.051,149.052
C06215=1165.185,23.520,-47.771,-179.882,6.052,149.052
C06216=1165.179,23.770,-47.786,-179.880,6.052,149.051
C06217=1165.175,24.019,-47.800,-179.877,6.053,149.051
C06218=1165.170,24.269,-47.815,-179.875,6.054,149.050
C06219=1165.165,24.518,-47.830,-179.872,6.055,149.049
C06220=1165.160,24.768,-47.844,-179.869,6.056,149.049
C06221=1165.155,25.018,-47.858,-179.867,6.057,149.048
C06222=1165.150,25.267,-47.874,-179.865,6.057,149.048
C06223=1165.145,25.517,-47.888,-179.862,6.058,149.047
C06224=1165.140,25.766,-47.902,-179.859,6.059,149.046
C06225=1165.135,26.015,-47.917,-179.857,6.060,149.046
C06226=1165.129,26.265,-47.932,-179.854,6.060,149.045
C06227=1165.124,26.514,-47.946,-179.852,6.061,149.045
C06228=1165.119,26.764,-47.961,-179.850,6.062,149.044
C06229=1165.114,27.013,-47.975,-179.846,6.063,149.044
C06230=1165.109,27.263,-47.990,-179.844,6.064,149.043
C06231=1165.104,27.512,-48.005,-179.842,6.064,149.042
C06232=1165.099,27.781,-48.021,-179.838,6.066,149.042
C06233=1165.094,28.050,-48.037,-179.836,6.067,149.041
C06234=1165.088,28.319,-48.053,-179.833,6.067,149.041
C06235=1165.083,28.588,-48.069,-179.830,6.068,149.040
C06236=1165.078,28.838,-48.083,-179.828,6.069,149.039
C06237=1165.072,29.088,-48.098,-179.825,6.070,149.039
C06238=1165.067,29.337,-48.113,-179.823,6.070,149.038
C06239=1165.062,29.586,-48.127,-179.820,6.072,149.038
C06240=1165.057,29.836,-48.143,-179.818,6.073,149.037
C06241=1165.052,30.085,-48.157,-179.815,6.073,149.037
C06242=1165.047,30.335,-48.172,-179.813,6.074,149.036
C06243=1165.042,30.585,-48.187,-179.810,6.075,149.035
C06244=1165.037,30.834,-48.202,-179.807,6.076,149.035
C06245=1165.032,31.083,-48.216,-179.805,6.077,149.034
C06246=1165.027,31.333,-48.232,-179.802,6.077,149.034
C06247=1165.022,31.583,-48.246,-179.800,6.079,149.033
C06248=1165.017,31.832,-48.261,-179.797,6.079,149.032
C06249=1165.011,32.082,-48.276,-179.795,6.080,149.032
C06250=1165.007,32.331,-48.291,-179.792,6.080,149.031
C06251=1165.002,32.580,-48.305,-179.789,6.082,149.031
C06252=1164.996,32.830,-48.321,-179.787,6.083,149.030
C06253=1164.992,33.079,-48.336,-179.784,6.083,149.030
C06254=1164.987,33.329,-48.350,-179.782,6.084,149.029
C06255=1164.981,33.578,-48.365,-179.779,6.085,149.028
C06256=1164.976,33.828,-48.380,-179.777,6.086,149.028
C06257=1164.971,34.077,-48.395,-179.774,6.087,149.027
C06258=1164.966,34.326,-48.410,-179.771,6.088,149.027
C06259=1164.961,34.576,-48.425,-179.769,6.089,149.026
C06260=1164.956,34.825,-48.440,-179.766,6.090,149.026
C06261=1164.952,35.075,-48.455,-179.764,6.090,149.025
C06262=1164.946,35.325,-48.470,-179.761,6.092,149.025
C06263=1164.942,35.574,-48.485,-179.758,6.092,149.024
C06264=1164.936,35.824,-48.501,-179.756,6.093,149.023
C06265=1164.931,36.073,-48.515,-179.754,6.093,149.023
C06266=1164.926,36.323,-48.531,-179.751,6.095,149.022
C06267=1164.921,36.572,-48.546,-179.748,6.096,149.022
C06268=1164.916,36.822,-48.561,-179.746,6.096,149.021
C06269=1164.911,37.071,-48.576,-179.743,6.098,149.021
C06270=1164.906,37.320,-48.591,-179.740,6.098,149.020
C06271=1164.901,37.569,-48.606,-179.738,6.099,149.019
C06272=1164.896,37.820,-48.621,-179.735,6.100,149.019
C06273=1164.891,38.069,-48.636,-179.733,6.101,149.018
C06274=1164.886,38.319,-48.652,-179.730,6.102,149.018
C06275=1164.881,38.568,-48.667,-179.728,6.103,149.017
C06276=1164.875,38.818,-48.682,-179.725,6.104,149.017
C06277=1164.871,39.067,-48.697,-179.722,6.105,149.016
C06278=1164.865,39.316,-48.713,-179.720,6.105,149.015
C06279=1164.861,39.566,-48.728,-179.718,6.106,149.015
C06280=1164.856,39.815,-48.743,-179.714,6.107,149.014
C06281=1164.850,40.066,-48.758,-179.712,6.108,149.014
C06282=1164.846,40.315,-48.773,-179.710,6.109,149.013
C06283=1164.840,40.564,-48.789,-179.707,6.110,149.013
C06284=1164.836,40.813,-48.804,-179.704,6.111,149.012
C06285=1164.831,41.063,-48.820,-179.702,6.112,149.012
C06286=1164.825,41.313,-48.835,-179.699,6.113,149.011
C06287=1164.821,41.562,-48.850,-179.697,6.114,149.010
C06288=1164.815,41.811,-48.866,-179.694,6.114,149.010
C06289=1164.810,42.061,-48.880,-179.691,6.116,149.009
C06290=1164.805,42.310,-48.896,-179.689,6.116,149.009
C06291=1164.800,42.560,-48.912,-179.686,6.117,149.008
C06292=1164.796,42.809,-48.927,-179.683,6.119,149.008
C06293=1164.790,43.059,-48.942,-179.681,6.119,149.007
C06294=1164.785,43.308,-48.958,-179.678,6.120,149.006
C06295=1164.781,43.558,-48.973,-179.676,6.120,149.006
C06296=1164.775,43.807,-48.989,-179.673,6.122,149.005
C06297=1164.770,44.057,-49.005,-179.670,6.123,149.005
C06298=1164.765,44.306,-49.020,-179.668,6.123,149.004
C06299=1164.760,44.555,-49.035,-179.665,6.125,149.004
C06300=1164.755,44.805,-49.051,-179.663,6.126,149.003
C06301=1164.751,45.054,-49.066,-179.660,6.126,149.002
C06302=1164.745,45.304,-49.082,-179.657,6.128,149.002
C06303=1164.740,45.553,-49.097,-179.655,6.128,149.001
C06304=1164.736,45.803,-49.113,-179.653,6.129,149.001
C06305=1164.730,46.053,-49.128,-179.649,6.130,149.000
C06306=1164.725,46.302,-49.144,-179.647,6.131,149.000
C06307=1164.720,46.551,-49.159,-179.645,6.132,148.999
C06308=1164.716,46.801,-49.175,-179.642,6.133,148.999
C06309=1164.710,47.050,-49.191,-179.639,6.134,148.998
C06310=1164.705,47.299,-49.207,-179.636,6.136,148.998
C06311=1164.700,47.549,-49.223,-179.634,6.136,148.997
C06312=1164.696,47.798,-49.238,-179.632,6.137,148.996
C06313=1164.690,48.048,-49.253,-179.628,6.138,148.996
C06314=1164.685,48.298,-49.269,-179.626,6.139,148.995
C06315=1164.680,48.547,-49.285,-179.624,6.140,148.995
C06316=1164.675,48.796,-49.300,-179.621,6.141,148.994
C06317=1164.670,49.045,-49.316,-179.618,6.142,148.994
C06318=1164.666,49.295,-49.332,-179.616,6.143,148.993
C06319=1164.660,49.545,-49.348,-179.613,6.144,148.992
C06320=1164.655,49.794,-49.363,-179.611,6.145,148.992
C06321=1164.651,50.044,-49.378,-179.608,6.145,148.991
C06322=1164.646,50.293,-49.395,-179.605,6.147,148.991
C06323=1164.640,50.542,-49.410,-179.603,6.147,148.990
C06324=1164.635,50.792,-49.426,-179.600,6.149,148.990
C06325=1164.630,51.042,-49.442,-179.597,6.150,148.989
C06326=1164.625,51.292,-49.458,-179.595,6.150,148.989
C06327=1164.621,51.540,-49.474,-179.592,6.152,148.988
C06328=1164.616,51.790,-49.489,-179.590,6.153,148.988
C06329=1164.611,52.040,-49.505,-179.587,6.153,148.987
C06330=1164.606,52.289,-49.521,-179.584,6.155,148.986
C06331=1164.600,52.538,-49.537,-179.582,6.156,148.986
C06332=1164.596,52.788,-49.553,-179.579,6.157,148.985
C06333=1164.590,53.037,-49.569,-179.577,6.158,148.985
C06334=1164.585,53.286,-49.585,-179.574,6.158,148.984
C06335=1164.580,53.536,-49.601,-179.571,6.160,148.984
C06336=1164.575,53.805,-49.618,-179.569,6.160,148.983
C06337=1164.569,54.073,-49.635,-179.566,6.162,148.982
C06338=1164.564,54.342,-49.652,-179.563,6.163,148.982
C06339=1164.559,54.610,-49.670,-179.560,6.164,148.981
C06340=1164.554,54.859,-49.685,-179.558,6.164,148.981
C06341=1164.550,55.110,-49.701,-179.555,6.166,148.980
C06342=1164.544,55.358,-49.717,-179.552,6.167,148.980
C06343=1164.539,55.608,-49.733,-179.549,6.168,148.979
C06344=1164.535,55.857,-49.749,-179.547,6.169,148.979
C06345=1164.529,56.107,-49.765,-179.545,6.170,148.978
C06346=1164.524,56.357,-49.781,-179.542,6.171,148.978
C06347=1164.519,56.605,-49.797,-179.539,6.172,148.977
C06348=1164.515,56.856,-49.813,-179.537,6.174,148.976
C06349=1164.509,57.104,-49.830,-179.534,6.174,148.976
C06350=1164.505,57.354,-49.846,-179.531,6.176,148.975
C06351=1164.500,57.603,-49.862,-179.529,6.176,148.975
C06352=1164.494,57.853,-49.877,-179.526,6.177,148.974
C06353=1164.490,58.102,-49.894,-179.523,6.178,148.974
C06354=1164.484,58.352,-49.910,-179.521,6.179,148.973
C06355=1164.479,58.601,-49.927,-179.518,6.181,148.972
C06356=1164.474,58.851,-49.943,-179.516,6.181,148.972
C06357=1164.469,59.100,-49.959,-179.513,6.182,148.971
C06358=1164.464,59.350,-49.975,-179.510,6.184,148.971
C06359=1164.459,59.599,-49.991,-179.508,6.184,148.970
C06360=1164.454,59.848,-50.008,-179.505,6.186,148.970
C06361=1164.450,60.098,-50.024,-179.503,6.187,148.969
C06362=1164.444,60.347,-50.040,-179.499,6.188,148.969
C06363=1164.440,60.597,-50.056,-179.497,6.189,148.968
C06364=1164.435,60.846,-50.072,-179.495,6.189,148.968
C06365=1164.430,61.095,-50.089,-179.492,6.191,148.967
C06366=1164.425,61.345,-50.105,-179.489,6.191,148.967
C06367=1164.419,61.594,-50.122,-179.487,6.193,148.966
C06368=1164.414,61.844,-50.137,-179.484,6.194,148.965
C06369=1164.410,62.093,-50.154,-179.481,6.195,148.965
C06370=1164.405,62.343,-50.171,-179.479,6.196,148.964
C06371=1164.400,62.592,-50.186,-179.476,6.198,148.964
C06372=1164.395,62.842,-50.203,-179.474,6.198,148.963
C06373=1164.390,63.090,-50.219,-179.471,6.199,148.963
C06374=1164.385,63.340,-50.237,-179.468,6.201,148.962
C06375=1164.380,63.590,-50.252,-179.466,6.201,148.962
C06376=1164.375,63.839,-50.269,-179.463,6.203,148.961
C06377=1164.370,64.088,-50.285,-179.460,6.203,148.961
C06378=1164.365,64.338,-50.301,-179.458,6.205,148.960
C06379=1164.360,64.588,-50.318,-179.455,6.205,148.960
C06380=1164.355,64.837,-50.335,-179.452,6.207,148.959
C06381=1164.350,65.086,-50.351,-179.450,6.208,148.959
C06382=1164.345,65.335,-50.367,-179.447,6.209,148.958
C06383=1164.341,65.585,-50.384,-179.445,6.210,148.958
C06384=1164.335,65.835,-50.401,-179.441,6.211,148.957
C06385=1164.330,66.083,-50.417,-179.439,6.212,148.956
C06386=1164.326,66.333,-50.434,-179.437,6.213,148.956
C06387=1164.321,66.582,-50.450,-179.434,6.215,148.955
C06388=1164.315,66.832,-50.467,-179.431,6.215,148.955
C06389=1164.311,67.082,-50.483,-179.429,6.217,148.954
C06390=1164.306,67.330,-50.500,-179.426,6.218,148.954
C06391=1164.301,67.580,-50.516,-179.423,6.219,148.953
C06392=1164.296,67.830,-50.534,-179.421,6.220,148.953
C06393=1164.291,68.078,-50.550,-179.418,6.221,148.952
C06394=1164.286,68.328,-50.567,-179.416,6.222,148.952
C06395=1164.281,68.578,-50.584,-179.412,6.223,148.951
C06396=1164.276,68.827,-50.599,-179.410,6.224,148.951
C06397=1164.271,69.077,-50.616,-179.408,6.226,148.950
C06398=1164.266,69.326,-50.633,-179.405,6.226,148.949
C06399=1164.261,69.575,-50.650,-179.402,6.228,148.949
C06400=1164.257,69.825,-50.666,-179.400,6.229,148.948
C06401=1164.251,70.075,-50.684,-179.397,6.230,148.948
C06402=1164.246,70.323,-50.700,-179.394,6.231,148.947
C06403=1164.242,70.573,-50.717,-179.391,6.232,148.947
C06404=1164.237,70.823,-50.734,-179.389,6.233,148.946
C06405=1164.231,71.071,-50.750,-179.386,6.235,148.946
C06406=1164.227,71.321,-50.767,-179.384,6.235,148.945
C06407=1164.222,71.571,-50.784,-179.381,6.237,148.945
C06408=1164.217,71.819,-50.800,-179.379,6.238,148.944
C06409=1164.211,72.069,-50.818,-179.375,6.239,148.944
C06410=1164.207,72.319,-50.834,-179.373,6.240,148.943
C06411=1164.202,72.568,-50.852,-179.371,6.242,148.943
C06412=1164.197,72.817,-50.868,-179.368,6.242,148.942
C06413=1164.192,73.067,-50.884,-179.365,6.244,148.942
C06414=1164.187,73.316,-50.902,-179.363,6.244,148.941
C06415=1164.183,73.565,-50.919,-179.360,6.246,148.941
C06416=1164.177,73.814,-50.936,-179.358,6.247,148.940
C06417=1164.173,74.064,-50.953,-179.354,6.248,148.939
C06418=1164.167,74.314,-50.970,-179.352,6.249,148.939
C06419=1164.163,74.563,-50.987,-179.349,6.250,148.938
C06420=1164.157,74.812,-51.004,-179.347,6.251,148.938
C06421=1164.153,75.062,-51.020,-179.344,6.253,148.938
C06422=1164.148,75.311,-51.038,-179.341,6.254,148.937
C06423=1164.143,75.561,-51.055,-179.339,6.255,148.936
C06424=1164.137,75.810,-51.072,-179.336,6.256,148.936
C06425=1164.133,76.059,-51.088,-179.333,6.257,148.935
C06426=1164.128,76.309,-51.106,-179.331,6.259,148.935
C06427=1164.123,76.558,-51.123,-179.328,6.260,148.934
C06428=1164.118,76.808,-51.140,-179.325,6.261,148.934
C06429=1164.113,77.056,-51.157,-179.323,6.262,148.933
C06430=1164.108,77.306,-51.174,-179.320,6.263,148.933
C06431=1164.104,77.555,-51.191,-179.318,6.264,148.932
C06432=1164.099,77.805,-51.209,-179.315,6.266,148.932
C06433=1164.094,78.054,-51.225,-179.312,6.266,148.931
C06434=1164.088,78.303,-51.242,-179.309,6.268,148.931
C06435=1164.083,78.553,-51.260,-179.307,6.270,148.930
C06436=1164.079,78.802,-51.277,-179.304,6.270,148.930
C06437=1164.074,79.052,-51.294,-179.301,6.272,148.929
C06438=1164.069,79.301,-51.311,-179.299,6.273,148.929
C06439=1164.064,79.550,-51.329,-179.296,6.274,148.928
C06440=1164.058,79.819,-51.347,-179.293,6.276,148.928
C06441=1164.054,80.087,-51.365,-179.290,6.276,148.927
C06442=1164.048,80.355,-51.385,-179.288,6.278,148.927
C06443=1164.043,80.624,-51.403,-179.285,6.279,148.926
C06444=1164.038,80.873,-51.420,-179.282,6.280,148.925
C06445=1164.033,81.122,-51.437,-179.279,6.281,148.925
C06446=1164.028,81.372,-51.455,-179.276,6.283,148.924
C06447=1164.024,81.621,-51.472,-179.274,6.284,148.924
C06448=1164.019,81.871,-51.489,-179.271,6.285,148.923
C06449=1164.013,82.121,-51.507,-179.269,6.286,148.923
C06450=1164.009,82.369,-51.524,-179.266,6.288,148.922
C06451=1164.003,82.618,-51.541,-179.264,6.288,148.922
C06452=1163.998,82.868,-51.559,-179.261,6.290,148.921
C06453=1163.993,83.117,-51.576,-179.258,6.291,148.921
C06454=1163.989,83.366,-51.594,-179.255,6.292,148.920
C06455=1163.984,83.616,-51.611,-179.253,6.294,148.920
C06456=1163.979,83.865,-51.629,-179.250,6.294,148.919
C06457=1163.974,84.115,-51.645,-179.247,6.296,148.919
C06458=1163.969,84.364,-51.663,-179.245,6.298,148.918
C06459=1163.964,84.614,-51.681,-179.242,6.298,148.918
C06460=1163.959,84.863,-51.699,-179.239,6.300,148.917
C06461=1163.955,85.112,-51.715,-179.237,6.301,148.917
C06462=1163.950,85.362,-51.733,-179.234,6.302,148.916
C06463=1163.945,85.611,-51.751,-179.231,6.304,148.916
C06464=1163.940,85.861,-51.769,-179.229,6.304,148.915
C06465=1163.935,86.110,-51.787,-179.226,6.306,148.915
C06466=1163.930,86.359,-51.803,-179.224,6.307,148.914
C06467=1163.925,86.608,-51.821,-179.221,6.308,148.914
C06468=1163.920,86.857,-51.839,-179.218,6.310,148.913
C06469=1163.915,87.107,-51.856,-179.216,6.311,148.913
C06470=1163.910,87.356,-51.874,-179.212,6.312,148.912
C06471=1163.906,87.605,-51.891,-179.210,6.313,148.912
C06472=1163.900,87.854,-51.909,-179.208,6.315,148.911
C06473=1163.896,88.104,-51.927,-179.204,6.316,148.911
C06474=1163.891,88.353,-51.945,-179.202,6.317,148.910
C06475=1163.885,88.603,-51.962,-179.199,6.319,148.910
C06476=1163.881,88.852,-51.980,-179.196,6.320,148.909
C06477=1163.876,89.101,-51.998,-179.194,6.321,148.909
C06478=1163.871,89.350,-52.015,-179.191,6.322,148.908
C06479=1163.866,89.600,-52.033,-179.189,6.323,148.908
C06480=1163.862,89.850,-52.051,-179.186,6.325,148.907
C06481=1163.857,90.099,-52.069,-179.183,6.326,148.907
C06482=1163.852,90.349,-52.086,-179.181,6.327,148.906
C06483=1163.847,90.598,-52.104,-179.178,6.329,148.906
C06484=1163.842,90.847,-52.122,-179.175,6.330,148.905
C06485=1163.837,91.096,-52.140,-179.173,6.331,148.905
C06486=1163.832,91.345,-52.158,-179.170,6.333,148.904
C06487=1163.827,91.595,-52.175,-179.167,6.333,148.904
C06488=1163.822,91.844,-52.193,-179.165,6.335,148.903
C06489=1163.817,92.093,-52.211,-179.162,6.337,148.903
C06490=1163.813,92.342,-52.229,-179.159,6.337,148.902
C06491=1163.808,92.591,-52.247,-179.156,6.339,148.902
C06492=1163.803,92.841,-52.265,-179.154,6.341,148.901
C06493=1163.798,93.090,-52.283,-179.151,6.341,148.901
C06494=1163.793,93.340,-52.300,-179.148,6.343,148.900
C06495=1163.789,93.589,-52.318,-179.146,6.345,148.900
C06496=1163.784,93.839,-52.336,-179.143,6.345,148.899
C06497=1163.779,94.088,-52.354,-179.140,6.347,148.899
C06498=1163.774,94.337,-52.372,-179.138,6.348,148.898
C06499=1163.769,94.586,-52.390,-179.135,6.349,148.898
C06500=1163.764,94.835,-52.408,-179.132,6.351,148.897
C06501=1163.758,95.085,-52.427,-179.130,6.352,148.897
C06502=1163.754,95.334,-52.445,-179.127,6.353,148.896
C06503=1163.749,95.583,-52.463,-179.124,6.355,148.896
C06504=1163.744,95.833,-52.481,-179.121,6.356,148.895
C06505=1163.739,96.082,-52.499,-179.119,6.357,148.895
C06506=1163.734,96.331,-52.517,-179.116,6.359,148.894
C06507=1163.730,96.581,-52.535,-179.113,6.360,148.894
C06508=1163.725,96.830,-52.553,-179.111,6.361,148.894
C06509=1163.720,97.079,-52.571,-179.108,6.363,148.893
C06510=1163.715,97.329,-52.589,-179.105,6.364,148.892
C06511=1163.711,97.578,-52.607,-179.103,6.365,148.892
C06512=1163.706,97.827,-52.625,-179.100,6.367,148.892
C06513=1163.700,98.077,-52.644,-179.097,6.368,148.891
C06514=1163.695,98.326,-52.662,-179.095,6.369,148.891
C06515=1163.690,98.575,-52.680,-179.092,6.371,148.890
C06516=1163.686,98.825,-52.698,-179.089,6.372,148.890
C06517=1163.681,99.073,-52.717,-179.086,6.374,148.889
C06518=1163.676,99.323,-52.735,-179.084,6.375,148.889
C06519=1163.671,99.572,-52.753,-179.081,6.376,148.888
C06520=1163.666,99.822,-52.772,-179.078,6.378,148.888
C06521=1163.661,100.071,-52.790,-179.076,6.379,148.887
C06522=1163.657,100.320,-52.808,-179.074,6.380,148.887
C06523=1163.652,100.569,-52.826,-179.070,6.382,148.886
C06524=1163.647,100.818,-52.844,-179.068,6.383,148.886
C06525=1163.642,101.068,-52.863,-179.065,6.384,148.885
C06526=1163.637,101.317,-52.881,-179.062,6.386,148.885
C06527=1163.632,101.567,-52.899,-179.060,6.387,148.884
C06528=1163.628,101.815,-52.918,-179.057,6.388,148.884
C06529=1163.623,102.065,-52.936,-179.055,6.390,148.883
C06530=1163.618,102.314,-52.955,-179.052,6.391,148.883
C06531=1163.613,102.564,-52.973,-179.049,6.392,148.882
C06532=1163.608,102.812,-52.992,-179.047,6.394,148.882
C06533=1163.604,103.062,-53.010,-179.043,6.395,148.881
C06534=1163.598,103.312,-53.028,-179.041,6.397,148.881
C06535=1163.593,103.560,-53.047,-179.039,6.398,148.881
C06536=1163.589,103.810,-53.066,-179.036,6.400,148.880
C06537=1163.584,104.059,-53.084,-179.033,6.401,148.879
C06538=1163.579,104.308,-53.103,-179.030,6.403,148.879
C06539=1163.574,104.557,-53.121,-179.028,6.403,148.879
C06540=1163.570,104.807,-53.139,-179.025,6.405,148.878
C06541=1163.564,105.056,-53.158,-179.022,6.407,148.878
C06542=1163.559,105.305,-53.176,-179.020,6.407,148.877
C06543=1163.555,105.555,-53.195,-179.017,6.409,148.877
C06544=1163.550,105.823,-53.215,-179.014,6.410,148.876
C06545=1163.545,106.091,-53.235,-179.011,6.412,148.876
C06546=1163.539,106.360,-53.255,-179.008,6.414,148.875
C06547=1163.534,106.628,-53.276,-179.005,6.415,148.875
C06548=1163.529,106.878,-53.294,-179.002,6.417,148.874
C06549=1163.524,107.126,-53.313,-179.000,6.419,148.874
C06550=1163.519,107.376,-53.332,-178.997,6.419,148.873
C06551=1163.514,107.626,-53.350,-178.994,6.421,148.873
C06552=1163.510,107.874,-53.368,-178.992,6.423,148.872
C06553=1163.505,108.124,-53.387,-178.989,6.424,148.872
C06554=1163.500,108.373,-53.406,-178.986,6.425,148.871
C06555=1163.495,108.623,-53.425,-178.984,6.427,148.871
C06556=1163.490,108.872,-53.443,-178.981,6.428,148.871
C06557=1163.485,109.120,-53.463,-178.978,6.430,148.870
C06558=1163.481,109.370,-53.481,-178.976,6.431,148.870
C06559=1163.476,109.619,-53.500,-178.973,6.432,148.869
C06560=1163.471,109.869,-53.519,-178.970,6.434,148.869
C06561=1163.466,110.118,-53.537,-178.967,6.436,148.868
C06562=1163.461,110.367,-53.556,-178.965,6.436,148.868
C06563=1163.457,110.616,-53.575,-178.962,6.438,148.867
C06564=1163.451,110.865,-53.594,-178.959,6.440,148.867
C06565=1163.447,111.115,-53.613,-178.957,6.441,148.866
C06566=1163.442,111.364,-53.632,-178.953,6.443,148.866
C06567=1163.437,111.613,-53.651,-178.951,6.444,148.865
C06568=1163.432,111.863,-53.670,-178.949,6.445,148.865
C06569=1163.428,112.111,-53.688,-178.946,6.447,148.865
C06570=1163.423,112.361,-53.707,-178.943,6.449,148.864
C06571=1163.418,112.610,-53.726,-178.941,6.449,148.864
C06572=1163.413,112.860,-53.746,-178.938,6.451,148.863
C06573=1163.408,113.108,-53.765,-178.935,6.453,148.863
C06574=1163.404,113.358,-53.783,-178.932,6.454,148.862
C06575=1163.398,113.607,-53.803,-178.929,6.456,148.862
C06576=1163.394,113.856,-53.821,-178.927,6.457,148.861
C06577=1163.389,114.106,-53.840,-178.924,6.458,148.861
C06578=1163.384,114.354,-53.859,-178.922,6.460,148.860
C06579=1163.379,114.604,-53.879,-178.919,6.462,148.860
C06580=1163.374,114.853,-53.898,-178.916,6.463,148.859
C06581=1163.370,115.102,-53.917,-178.914,6.464,148.859
C06582=1163.364,115.352,-53.935,-178.911,6.466,148.859
C06583=1163.359,115.601,-53.955,-178.908,6.468,148.858
C06584=1163.355,115.850,-53.974,-178.905,6.469,148.858
C06585=1163.350,116.099,-53.993,-178.902,6.471,148.857
C06586=1163.345,116.348,-54.012,-178.900,6.472,148.857
C06587=1163.341,116.597,-54.032,-178.897,6.473,148.856
C06588=1163.335,116.847,-54.050,-178.895,6.475,148.856
C06589=1163.331,117.096,-54.069,-178.892,6.477,148.856
C06590=1163.326,117.346,-54.089,-178.889,6.478,148.855
C06591=1163.321,117.595,-54.108,-178.886,6.480,148.855
C06592=1163.316,117.844,-54.128,-178.884,6.481,148.854
C06593=1163.312,118.093,-54.147,-178.881,6.482,148.854
C06594=1163.307,118.342,-54.166,-178.879,6.484,148.853
C06595=1163.302,118.591,-54.186,-178.875,6.485,148.853
C06596=1163.298,118.840,-54.205,-178.873,6.487,148.852
C06597=1163.292,119.089,-54.224,-178.870,6.489,148.852
C06598=1163.287,119.339,-54.244,-178.868,6.490,148.851
C06599=1163.283,119.588,-54.263,-178.865,6.491,148.851
C06600=1163.278,119.837,-54.282,-178.862,6.493,148.850
C06601=1163.273,120.087,-54.302,-178.859,6.495,148.850
C06602=1163.268,120.335,-54.321,-178.856,6.496,148.850
C06603=1163.263,120.585,-54.341,-178.854,6.498,148.849
C06604=1163.259,120.834,-54.360,-178.852,6.499,148.849
C06605=1163.254,121.083,-54.379,-178.849,6.501,148.848
C06606=1163.249,121.333,-54.399,-178.846,6.502,148.848
C06607=1163.244,121.582,-54.418,-178.843,6.504,148.847
C06608=1163.239,121.831,-54.438,-178.840,6.505,148.847
C06609=1163.235,122.080,-54.457,-178.838,6.507,148.847
C06610=1163.230,122.329,-54.476,-178.835,6.509,148.846
C06611=1163.225,122.579,-54.496,-178.833,6.510,148.846
C06612=1163.220,122.828,-54.515,-178.830,6.511,148.845
C06613=1163.215,123.077,-54.535,-178.827,6.513,148.845
C06614=1163.211,123.326,-54.554,-178.824,6.515,148.844
C06615=1163.206,123.576,-54.574,-178.821,6.516,148.844
C06616=1163.201,123.824,-54.593,-178.819,6.518,148.844
C06617=1163.196,124.074,-54.613,-178.816,6.520,148.843
C06618=1163.192,124.324,-54.633,-178.813,6.520,148.843
C06619=1163.186,124.572,-54.652,-178.811,6.522,148.842
C06620=1163.182,124.821,-54.672,-178.808,6.524,148.842
C06621=1163.177,125.071,-54.692,-178.805,6.525,148.841
C06622=1163.173,125.319,-54.711,-178.803,6.527,148.841
C06623=1163.168,125.569,-54.730,-178.800,6.529,148.841
C06624=1163.163,125.818,-54.751,-178.797,6.531,148.840
C06625=1163.158,126.067,-54.770,-178.794,6.532,148.840
C06626=1163.153,126.316,-54.790,-178.791,6.534,148.839
C06627=1163.149,126.566,-54.809,-178.789,6.535,148.839
C06628=1163.144,126.815,-54.830,-178.786,6.536,148.838
C06629=1163.139,127.064,-54.849,-178.784,6.538,148.838
C06630=1163.134,127.313,-54.869,-178.781,6.540,148.838
C06631=1163.130,127.562,-54.889,-178.778,6.542,148.837
C06632=1163.124,127.811,-54.908,-178.775,6.543,148.837
C06633=1163.119,128.061,-54.928,-178.772,6.545,148.836
C06634=1163.115,128.310,-54.948,-178.770,6.546,148.836
C06635=1163.110,128.559,-54.968,-178.767,6.548,148.835
C06636=1163.105,128.808,-54.987,-178.765,6.549,148.835
C06637=1163.100,129.057,-55.008,-178.762,6.551,148.835
C06638=1163.096,129.307,-55.027,-178.759,6.552,148.834
C06639=1163.091,129.556,-55.048,-178.757,6.554,148.834
C06640=1163.086,129.804,-55.067,-178.753,6.556,148.833
C06641=1163.081,130.054,-55.087,-178.751,6.557,148.833
C06642=1163.077,130.303,-55.107,-178.748,6.559,148.832
C06643=1163.072,130.553,-55.127,-178.745,6.561,148.832
C06644=1163.068,130.801,-55.147,-178.743,6.562,148.832
C06645=1163.062,131.050,-55.166,-178.740,6.564,148.831
C06646=1163.058,131.299,-55.187,-178.737,6.566,148.831
C06647=1163.052,131.549,-55.207,-178.735,6.568,148.830
C06648=1163.048,131.817,-55.229,-178.731,6.569,148.830
C06649=1163.043,132.086,-55.250,-178.729,6.571,148.829
C06650=1163.037,132.355,-55.271,-178.726,6.572,148.829
C06651=1163.033,132.623,-55.293,-178.723,6.574,148.829
C06652=1163.028,132.872,-55.313,-178.720,6.575,148.828
C06653=1163.023,133.122,-55.334,-178.717,6.577,148.828
C06654=1163.017,133.371,-55.353,-178.715,6.579,148.827
C06655=1163.013,133.619,-55.374,-178.712,6.581,148.827
C06656=1163.008,133.869,-55.393,-178.709,6.582,148.826
C06657=1163.004,134.118,-55.414,-178.706,6.584,148.826
C06658=1162.999,134.367,-55.434,-178.704,6.586,148.826
C06659=1162.994,134.617,-55.454,-178.701,6.588,148.825
C06660=1162.989,134.866,-55.475,-178.698,6.589,148.825
C06661=1162.984,135.114,-55.495,-178.696,6.591,148.825
C06662=1162.980,135.364,-55.514,-178.692,6.592,148.824
C06663=1162.975,135.613,-55.535,-178.690,6.593,148.823
C06664=1162.970,135.862,-55.556,-178.688,6.595,148.823
C06665=1162.965,136.111,-55.575,-178.685,6.597,148.823
C06666=1162.961,136.360,-55.596,-178.682,6.599,148.822
C06667=1162.956,136.609,-55.616,-178.680,6.600,148.822
C06668=1162.951,136.859,-55.636,-178.677,6.602,148.822
C06669=1162.946,137.108,-55.657,-178.674,6.604,148.821
C06670=1162.942,137.357,-55.677,-178.671,6.605,148.821
C06671=1162.937,137.605,-55.697,-178.669,6.607,148.820
C06672=1162.931,137.855,-55.717,-178.666,6.609,148.820
C06673=1162.927,138.104,-55.738,-178.663,6.611,148.820
C06674=1162.923,138.353,-55.758,-178.661,6.612,148.819
C06675=1162.917,138.602,-55.779,-178.658,6.614,148.819
C06676=1162.913,138.851,-55.799,-178.655,6.615,148.818
C06677=1162.909,139.100,-55.820,-178.652,6.617,148.818
C06678=1162.904,139.350,-55.839,-178.649,6.619,148.817
C06679=1162.899,139.599,-55.860,-178.647,6.621,148.817
C06680=1162.894,139.848,-55.881,-178.644,6.622,148.817
C06681=1162.890,140.097,-55.901,-178.641,6.624,148.816
C06682=1162.885,140.346,-55.922,-178.638,6.626,148.816
C06683=1162.880,140.595,-55.942,-178.636,6.628,148.815
C06684=1162.875,140.844,-55.963,-178.633,6.629,148.815
C06685=1162.871,141.093,-55.984,-178.630,6.631,148.815
C06686=1162.866,141.343,-56.003,-178.628,6.633,148.814
C06687=1162.861,141.592,-56.024,-178.625,6.635,148.814
C06688=1162.856,141.841,-56.045,-178.622,6.636,148.814
C06689=1162.852,142.090,-56.065,-178.620,6.638,148.813
C06690=1162.847,142.339,-56.086,-178.617,6.640,148.813
C06691=1162.842,142.588,-56.106,-178.614,6.641,148.812
C06692=1162.837,142.838,-56.127,-178.611,6.643,148.812
C06693=1162.832,143.087,-56.148,-178.609,6.645,148.812
C06694=1162.827,143.336,-56.169,-178.606,6.647,148.811
C06695=1162.823,143.585,-56.189,-178.603,6.648,148.811
C06696=1162.818,143.834,-56.209,-178.601,6.650,148.810
C06697=1162.813,144.083,-56.230,-178.598,6.652,148.810
C06698=1162.809,144.332,-56.251,-178.595,6.653,148.809
C06699=1162.804,144.581,-56.273,-178.592,6.655,148.809
C06700=1162.800,144.829,-56.293,-178.589,6.657,148.809
C06701=1162.794,145.079,-56.314,-178.587,6.658,148.808
C06702=1162.791,145.328,-56.335,-178.584,6.660,148.808
C06703=1162.785,145.578,-56.356,-178.581,6.662,148.808
C06704=1162.781,145.827,-56.376,-178.579,6.664,148.807
C06705=1162.776,146.076,-56.397,-178.576,6.665,148.807
C06706=1162.771,146.325,-56.417,-178.573,6.667,148.806
C06707=1162.766,146.574,-56.438,-178.570,6.669,148.806
C06708=1162.761,146.823,-56.460,-178.568,6.671,148.806
C06709=1162.757,147.072,-56.480,-178.565,6.672,148.805
C06710=1162.752,147.321,-56.501,-178.562,6.674,148.805
C06711=1162.747,147.570,-56.522,-178.560,6.676,148.804
C06712=1162.743,147.820,-56.543,-178.557,6.678,148.804
C06713=1162.738,148.068,-56.564,-178.554,6.679,148.804
C06714=1162.733,148.317,-56.585,-178.552,6.681,148.803
C06715=1162.728,148.567,-56.606,-178.548,6.684,148.803
C06716=1162.724,148.816,-56.626,-178.546,6.685,148.803
C06717=1162.719,149.064,-56.648,-178.543,6.687,148.802
C06718=1162.714,149.313,-56.668,-178.540,6.689,148.802
C06719=1162.709,149.562,-56.689,-178.537,6.690,148.801
C06720=1162.705,149.812,-56.711,-178.535,6.692,148.801
C06721=1162.701,150.061,-56.732,-178.532,6.694,148.801
C06722=1162.695,150.310,-56.753,-178.529,6.696,148.800
C06723=1162.690,150.559,-56.774,-178.527,6.697,148.800
C06724=1162.686,150.808,-56.795,-178.524,6.699,148.800
C06725=1162.681,151.057,-56.816,-178.521,6.701,148.799
C06726=1162.677,151.306,-56.838,-178.519,6.703,148.799
C06727=1162.672,151.555,-56.858,-178.516,6.704,148.798
C06728=1162.667,151.804,-56.879,-178.514,6.706,148.798
C06729=1162.662,152.053,-56.901,-178.511,6.708,148.798
C06730=1162.657,152.302,-56.922,-178.508,6.710,148.797
C06731=1162.653,152.551,-56.943,-178.506,6.712,148.797
C06732=1162.648,152.801,-56.964,-178.502,6.714,148.797
C06733=1162.643,153.049,-56.986,-178.500,6.716,148.796
C06734=1162.638,153.299,-57.007,-178.497,6.718,148.796
C06735=1162.634,153.548,-57.028,-178.494,6.719,148.796
C06736=1162.629,153.797,-57.049,-178.491,6.721,148.795
C06737=1162.624,154.046,-57.070,-178.489,6.723,148.795
C06738=1162.619,154.295,-57.092,-178.486,6.725,148.794
C06739=1162.615,154.544,-57.112,-178.483,6.726,148.794
C06740=1162.611,154.793,-57.134,-178.481,6.728,148.794
C06741=1162.606,155.042,-57.156,-178.478,6.730,148.793
C06742=1162.601,155.291,-57.177,-178.475,6.732,148.793
C06743=1162.596,155.540,-57.199,-178.472,6.734,148.793
C06744=1162.592,155.789,-57.219,-178.469,6.736,148.792
C06745=1162.587,156.038,-57.241,-178.467,6.738,148.792
C06746=1162.582,156.287,-57.262,-178.464,6.739,148.791
C06747=1162.578,156.536,-57.284,-178.461,6.741,148.791
C06748=1162.573,156.785,-57.306,-178.458,6.743,148.791
C06749=1162.568,157.034,-57.327,-178.456,6.745,148.790
C06750=1162.563,157.284,-57.349,-178.454,6.747,148.790
C06751=1162.559,157.532,-57.370,-178.451,6.749,148.790
C06752=1162.554,157.801,-57.393,-178.448,6.751,148.789
C06753=1162.549,158.070,-57.416,-178.444,6.752,148.789
C06754=1162.544,158.340,-57.439,-178.442,6.754,148.788
C06755=1162.539,158.608,-57.463,-178.438,6.757,148.788
C06756=1162.534,158.857,-57.484,-178.436,6.758,148.788
C06757=1162.529,159.106,-57.506,-178.433,6.760,148.787
C06758=1162.525,159.355,-57.528,-178.431,6.762,148.787
C06759=1162.520,159.604,-57.549,-178.428,6.764,148.787
C06760=1162.515,159.853,-57.570,-178.425,6.766,148.786
C06761=1162.510,160.103,-57.592,-178.422,6.768,148.786
C06762=1162.506,160.351,-57.614,-178.419,6.770,148.786
C06763=1162.501,160.600,-57.636,-178.417,6.772,148.785
C06764=1162.496,160.849,-57.658,-178.414,6.774,148.785
C06765=1162.491,161.099,-57.679,-178.411,6.775,148.785
C06766=1162.487,161.348,-57.701,-178.409,6.777,148.784
C06767=1162.482,161.597,-57.722,-178.406,6.779,148.784
C06768=1162.477,161.845,-57.744,-178.403,6.781,148.784
C06769=1162.473,162.095,-57.766,-178.401,6.784,148.783
C06770=1162.468,162.343,-57.788,-178.398,6.785,148.783
C06771=1162.464,162.593,-57.810,-178.395,6.787,148.783
C06772=1162.459,162.842,-57.831,-178.392,6.789,148.782
C06773=1162.454,163.090,-57.852,-178.390,6.790,148.782
C06774=1162.450,163.340,-57.875,-178.387,6.792,148.781
C06775=1162.445,163.588,-57.896,-178.384,6.795,148.781
C06776=1162.440,163.838,-57.918,-178.381,6.797,148.781
C06777=1162.436,164.086,-57.940,-178.378,6.798,148.780
C06778=1162.431,164.336,-57.962,-178.376,6.800,148.780
C06779=1162.426,164.584,-57.984,-178.373,6.802,148.780
C06780=1162.421,164.833,-58.006,-178.371,6.804,148.779
C06781=1162.417,165.083,-58.028,-178.368,6.806,148.779
C06782=1162.412,165.331,-58.050,-178.365,6.808,148.779
C06783=1162.407,165.581,-58.072,-178.362,6.810,148.778
C06784=1162.403,165.829,-58.093,-178.359,6.812,148.778
C06785=1162.398,166.079,-58.115,-178.357,6.813,148.778
C06786=1162.393,166.327,-58.137,-178.355,6.816,148.778
C06787=1162.389,166.577,-58.159,-178.351,6.818,148.777
C06788=1162.384,166.826,-58.181,-178.349,6.820,148.777
C06789=1162.379,167.075,-58.204,-178.346,6.822,148.776
C06790=1162.375,167.323,-58.226,-178.343,6.823,148.776
C06791=1162.370,167.572,-58.248,-178.340,6.825,148.776
C06792=1162.366,167.821,-58.270,-178.337,6.828,148.775
C06793=1162.361,168.071,-58.292,-178.335,6.830,148.775
C06794=1162.356,168.319,-58.314,-178.332,6.831,148.775
C06795=1162.351,168.569,-58.336,-178.330,6.833,148.774
C06796=1162.347,168.817,-58.358,-178.327,6.835,148.774
C06797=1162.342,169.066,-58.381,-178.324,6.838,148.774
C06798=1162.337,169.315,-58.403,-178.321,6.839,148.773
C06799=1162.333,169.564,-58.425,-178.318,6.841,148.773
C06800=1162.328,169.813,-58.446,-178.316,6.843,148.773
C06801=1162.323,170.062,-58.469,-178.313,6.845,148.772
C06802=1162.319,170.311,-58.492,-178.310,6.847,148.772
C06803=1162.314,170.560,-58.514,-178.307,6.849,148.772
C06804=1162.310,170.809,-58.536,-178.305,6.851,148.771
C06805=1162.304,171.058,-58.558,-178.302,6.853,148.771
C06806=1162.300,171.307,-58.581,-178.300,6.855,148.771
C06807=1162.295,171.555,-58.602,-178.297,6.857,148.771
C06808=1162.290,171.805,-58.625,-178.294,6.859,148.770
C06809=1162.286,172.054,-58.648,-178.291,6.861,148.770
C06810=1162.281,172.302,-58.669,-178.288,6.863,148.769
C06811=1162.276,172.552,-58.692,-178.286,6.864,148.769
C06812=1162.272,172.800,-58.714,-178.283,6.867,148.769
C06813=1162.268,173.049,-58.737,-178.280,6.869,148.769
C06814=1162.263,173.299,-58.759,-178.278,6.871,148.768
C06815=1162.258,173.547,-58.782,-178.275,6.873,148.768
C06816=1162.253,173.797,-58.804,-178.272,6.875,148.767
C06817=1162.249,174.046,-58.827,-178.269,6.877,148.767
C06818=1162.244,174.294,-58.849,-178.267,6.879,148.767
C06819=1162.240,174.543,-58.872,-178.264,6.881,148.767
C06820=1162.235,174.792,-58.894,-178.261,6.883,148.766
C06821=1162.230,175.042,-58.916,-178.258,6.885,148.766
C06822=1162.226,175.290,-58.939,-178.256,6.887,148.766
C06823=1162.221,175.539,-58.961,-178.253,6.889,148.765
C06824=1162.216,175.788,-58.984,-178.250,6.891,148.765
C06825=1162.212,176.037,-59.006,-178.247,6.893,148.765
C06826=1162.207,176.286,-59.030,-178.245,6.895,148.764
C06827=1162.202,176.535,-59.051,-178.242,6.897,148.764
C06828=1162.198,176.784,-59.075,-178.239,6.900,148.764
C06829=1162.194,177.033,-59.097,-178.236,6.901,148.763
C06830=1162.188,177.282,-59.120,-178.234,6.903,148.763
C06831=1162.184,177.530,-59.142,-178.232,6.905,148.763
C06832=1162.179,177.780,-59.165,-178.228,6.908,148.763
C06833=1162.174,178.028,-59.187,-178.226,6.910,148.762
C06834=1162.170,178.277,-59.211,-178.223,6.911,148.762
C06835=1162.165,178.526,-59.233,-178.220,6.913,148.762
C06836=1162.161,178.775,-59.256,-178.217,6.916,148.761
C06837=1162.156,179.024,-59.278,-178.215,6.918,148.761
C06838=1162.151,179.273,-59.301,-178.212,6.920,148.761
C06839=1162.147,179.522,-59.324,-178.209,6.921,148.760
C06840=1162.143,179.771,-59.347,-178.207,6.924,148.760
C06841=1162.137,180.020,-59.370,-178.204,6.926,148.760
C06842=1162.133,180.269,-59.392,-178.201,6.928,148.759
C06843=1162.128,180.518,-59.416,-178.198,6.930,148.759
C06844=1162.124,180.767,-59.438,-178.196,6.932,148.759
C06845=1162.119,181.015,-59.461,-178.193,6.934,148.759
C06846=1162.114,181.264,-59.484,-178.190,6.936,148.758
C06847=1162.110,181.513,-59.507,-178.187,6.939,148.758
C06848=1162.105,181.763,-59.530,-178.185,6.941,148.758
C06849=1162.101,182.011,-59.552,-178.182,6.942,148.757
C06850=1162.096,182.260,-59.575,-178.179,6.945,148.757
C06851=1162.091,182.509,-59.599,-178.176,6.947,148.757
C06852=1162.087,182.757,-59.621,-178.174,6.949,148.757
C06853=1162.082,183.006,-59.645,-178.171,6.951,148.756
C06854=1162.077,183.256,-59.667,-178.168,6.953,148.756
C06855=1162.073,183.504,-59.690,-178.165,6.955,148.756
C06856=1162.068,183.775,-59.715,-178.163,6.958,148.755
C06857=1162.063,184.044,-59.741,-178.160,6.960,148.755
C06858=1162.059,184.313,-59.765,-178.157,6.962,148.755
C06859=1162.053,184.583,-59.790,-178.154,6.964,148.754
C06860=1162.049,184.832,-59.814,-178.151,6.966,148.754
C06861=1162.043,185.080,-59.837,-178.148,6.968,148.754
C06862=1162.039,185.329,-59.860,-178.146,6.970,148.754
C06863=1162.035,185.578,-59.883,-178.143,6.973,148.753
C06864=1162.030,185.827,-59.906,-178.140,6.975,148.753
C06865=1162.025,186.076,-59.930,-178.138,6.977,148.753
C06866=1162.021,186.325,-59.952,-178.134,6.979,148.752
C06867=1162.017,186.574,-59.976,-178.132,6.981,148.752
C06868=1162.012,186.823,-59.999,-178.129,6.983,148.752
C06869=1162.007,187.071,-60.022,-178.126,6.986,148.752
C06870=1162.002,187.320,-60.046,-178.124,6.988,148.751
C06871=1161.998,187.569,-60.068,-178.121,6.989,148.751
C06872=1161.993,187.818,-60.092,-178.118,6.992,148.751
C06873=1161.988,188.067,-60.115,-178.115,6.994,148.750
C06874=1161.984,188.316,-60.138,-178.113,6.996,148.750
C06875=1161.979,188.565,-60.162,-178.110,6.999,148.750
C06876=1161.974,188.814,-60.185,-178.107,7.000,148.750
C06877=1161.970,189.063,-60.208,-178.105,7.002,148.749
C06878=1161.966,189.311,-60.232,-178.102,7.005,148.749
C06879=1161.961,189.560,-60.255,-178.099,7.007,148.749
C06880=1161.957,189.809,-60.279,-178.096,7.009,148.748
C06881=1161.952,190.058,-60.302,-178.094,7.012,148.748
C06882=1161.947,190.307,-60.325,-178.091,7.013,148.748
C06883=1161.942,190.556,-60.348,-178.088,7.015,148.748
C06884=1161.937,190.804,-60.372,-178.085,7.018,148.747
C06885=1161.933,191.053,-60.396,-178.083,7.020,148.747
C06886=1161.928,191.302,-60.419,-178.080,7.022,148.747
C06887=1161.923,191.551,-60.442,-178.077,7.024,148.747
C06888=1161.919,191.800,-60.467,-178.075,7.026,148.746
C06889=1161.914,192.049,-60.490,-178.071,7.029,148.746
C06890=1161.910,192.298,-60.513,-178.069,7.031,148.746
C06891=1161.905,192.547,-60.537,-178.066,7.033,148.745
C06892=1161.901,192.795,-60.561,-178.063,7.035,148.745
C06893=1161.896,193.044,-60.584,-178.061,7.037,148.745
C06894=1161.891,193.293,-60.607,-178.058,7.039,148.745
C06895=1161.887,193.542,-60.632,-178.055,7.042,148.744
C06896=1161.882,193.791,-60.655,-178.053,7.044,148.744
C06897=1161.877,194.040,-60.678,-178.050,7.046,148.744
C06898=1161.873,194.288,-60.702,-178.047,7.048,148.743
C06899=1161.869,194.538,-60.726,-178.045,7.050,148.743
C06900=1161.864,194.786,-60.750,-178.041,7.053,148.743
C06901=1161.860,195.035,-60.773,-178.039,7.055,148.743
C06902=1161.855,195.284,-60.797,-178.036,7.058,148.743
C06903=1161.851,195.533,-60.821,-178.033,7.059,148.742
C06904=1161.846,195.782,-60.844,-178.031,7.061,148.742
C06905=1161.842,196.030,-60.868,-178.028,7.064,148.742
C06906=1161.837,196.279,-60.892,-178.025,7.066,148.741
C06907=1161.832,196.528,-60.916,-178.022,7.069,148.741
C06908=1161.828,196.777,-60.939,-178.020,7.070,148.741
C06909=1161.823,197.025,-60.964,-178.017,7.072,148.741
C06910=1161.818,197.274,-60.987,-178.014,7.075,148.740
C06911=1161.814,197.523,-61.011,-178.012,7.077,148.740
C06912=1161.809,197.773,-61.035,-178.009,7.080,148.740
C06913=1161.805,198.021,-61.059,-178.006,7.082,148.740
C06914=1161.801,198.269,-61.083,-178.003,7.083,148.739
C06915=1161.796,198.518,-61.106,-178.001,7.086,148.739
C06916=1161.791,198.767,-61.131,-177.998,7.088,148.739
C06917=1161.786,199.016,-61.154,-177.995,7.091,148.739
C06918=1161.782,199.265,-61.179,-177.993,7.093,148.738
C06919=1161.778,199.514,-61.203,-177.990,7.095,148.738
C06920=1161.773,199.763,-61.226,-177.987,7.097,148.738
C06921=1161.768,200.012,-61.251,-177.984,7.099,148.738
C06922=1161.764,200.260,-61.275,-177.982,7.102,148.737
C06923=1161.759,200.509,-61.298,-177.979,7.104,148.737
C06924=1161.755,200.757,-61.323,-177.976,7.107,148.737
C06925=1161.750,201.007,-61.348,-177.973,7.109,148.737
C06926=1161.745,201.256,-61.371,-177.971,7.110,148.736
C06927=1161.741,201.504,-61.395,-177.968,7.113,148.736
C06928=1161.737,201.753,-61.419,-177.965,7.115,148.736
C06929=1161.731,202.001,-61.444,-177.963,7.118,148.736
C06930=1161.727,202.251,-61.467,-177.960,7.120,148.735
C06931=1161.723,202.500,-61.492,-177.957,7.122,148.735
C06932=1161.718,202.748,-61.516,-177.954,7.125,148.735
C06933=1161.713,202.997,-61.540,-177.951,7.127,148.735
C06934=1161.709,203.245,-61.564,-177.949,7.129,148.735
C06935=1161.705,203.495,-61.588,-177.946,7.131,148.734
C06936=1161.700,203.744,-61.613,-177.944,7.134,148.734
C06937=1161.695,203.992,-61.637,-177.941,7.136,148.734
C06938=1161.691,204.240,-61.661,-177.938,7.138,148.733
C06939=1161.686,204.490,-61.686,-177.935,7.140,148.733
C06940=1161.682,204.738,-61.710,-177.932,7.143,148.733
C06941=1161.677,204.987,-61.735,-177.930,7.145,148.733
C06942=1161.673,205.235,-61.759,-177.927,7.148,148.733
C06943=1161.669,205.484,-61.783,-177.924,7.150,148.732
C06944=1161.663,205.734,-61.807,-177.921,7.152,148.732
C06945=1161.659,205.982,-61.831,-177.919,7.154,148.732
C06946=1161.654,206.231,-61.856,-177.916,7.156,148.732
C06947=1161.650,206.480,-61.880,-177.914,7.159,148.732
C06948=1161.645,206.729,-61.905,-177.911,7.161,148.731
C06949=1161.640,206.977,-61.929,-177.908,7.164,148.731
C06950=1161.637,207.226,-61.954,-177.905,7.166,148.731
C06951=1161.632,207.475,-61.978,-177.902,7.168,148.730
C06952=1161.627,207.723,-62.002,-177.900,7.170,148.730
C06953=1161.623,207.973,-62.027,-177.897,7.173,148.730
C06954=1161.619,208.221,-62.052,-177.895,7.175,148.730
C06955=1161.613,208.469,-62.077,-177.891,7.178,148.730
C06956=1161.610,208.718,-62.101,-177.889,7.180,148.729
C06957=1161.604,208.967,-62.126,-177.886,7.182,148.729
C06958=1161.600,209.216,-62.150,-177.884,7.184,148.729
C06959=1161.596,209.465,-62.175,-177.880,7.187,148.729
C06960=1161.590,209.735,-62.202,-177.878,7.190,148.729
C06961=1161.585,210.005,-62.228,-177.875,7.192,148.728
C06962=1161.581,210.276,-62.255,-177.872,7.194,148.728
C06963=1161.576,210.546,-62.282,-177.869,7.197,148.728
C06964=1161.571,210.796,-62.307,-177.866,7.200,148.727
C06965=1161.567,211.044,-62.331,-177.863,7.202,148.727
C06966=1161.562,211.293,-62.356,-177.860,7.205,148.727
C06967=1161.558,211.542,-62.380,-177.858,7.207,148.727
C06968=1161.553,211.790,-62.406,-177.855,7.209,148.727
C06969=1161.548,212.040,-62.431,-177.853,7.211,148.726
C06970=1161.544,212.288,-62.455,-177.849,7.214,148.726
C06971=1161.539,212.536,-62.480,-177.847,7.216,148.726
C06972=1161.535,212.785,-62.505,-177.844,7.219,148.726
C06973=1161.530,213.034,-62.529,-177.842,7.221,148.726
C06974=1161.526,213.283,-62.554,-177.838,7.223,148.725
C06975=1161.522,213.531,-62.579,-177.836,7.226,148.725
C06976=1161.517,213.781,-62.604,-177.833,7.228,148.725
C06977=1161.512,214.029,-62.629,-177.831,7.230,148.725
C06978=1161.508,214.277,-62.654,-177.828,7.233,148.725
C06979=1161.503,214.527,-62.679,-177.825,7.235,148.724
C06980=1161.498,214.775,-62.704,-177.823,7.238,148.724
C06981=1161.494,215.024,-62.729,-177.820,7.240,148.724
C06982=1161.490,215.272,-62.753,-177.817,7.243,148.724
C06983=1161.485,215.521,-62.779,-177.814,7.244,148.723
C06984=1161.480,215.770,-62.804,-177.812,7.247,148.723
C06985=1161.477,216.019,-62.829,-177.808,7.250,148.723
C06986=1161.472,216.267,-62.853,-177.806,7.252,148.723
C06987=1161.467,216.516,-62.879,-177.803,7.255,148.723
C06988=1161.462,216.765,-62.904,-177.801,7.257,148.723
C06989=1161.458,217.014,-62.930,-177.798,7.260,148.722
C06990=1161.454,217.262,-62.954,-177.795,7.261,148.722
C06991=1161.449,217.511,-62.979,-177.792,7.264,148.722
C06992=1161.444,217.760,-63.004,-177.790,7.266,148.722
C06993=1161.440,218.008,-63.030,-177.787,7.269,148.722
C06994=1161.436,218.257,-63.054,-177.784,7.272,148.721
C06995=1161.431,218.506,-63.080,-177.782,7.274,148.721
C06996=1161.426,218.754,-63.104,-177.779,7.277,148.721
C06997=1161.422,219.003,-63.130,-177.776,7.279,148.721
C06998=1161.418,219.252,-63.156,-177.773,7.281,148.721
C06999=1161.413,219.501,-63.181,-177.771,7.283,148.720
C07000=1161.408,219.749,-63.206,-177.768,7.286,148.720
C07001=1161.404,219.997,-63.231,-177.765,7.288,148.720
C07002=1161.400,220.247,-63.256,-177.762,7.291,148.720
C07003=1161.395,220.495,-63.282,-177.760,7.294,148.720
C07004=1161.391,220.744,-63.307,-177.757,7.296,148.719
C07005=1161.386,220.993,-63.332,-177.754,7.299,148.719
C07006=1161.381,221.241,-63.358,-177.752,7.300,148.719
C07007=1161.377,221.490,-63.383,-177.749,7.303,148.719
C07008=1161.372,221.738,-63.409,-177.746,7.306,148.719
C07009=1161.368,221.987,-63.434,-177.743,7.308,148.718
C07010=1161.364,222.236,-63.460,-177.741,7.311,148.718
C07011=1161.359,222.484,-63.485,-177.738,7.313,148.718
C07012=1161.355,222.733,-63.511,-177.735,7.316,148.718
C07013=1161.349,222.982,-63.535,-177.732,7.319,148.718
C07014=1161.345,223.231,-63.561,-177.730,7.320,148.717
C07015=1161.341,223.479,-63.587,-177.727,7.323,148.717
C07016=1161.336,223.728,-63.612,-177.724,7.325,148.717
C07017=1161.332,223.976,-63.638,-177.722,7.328,148.717
C07018=1161.328,224.225,-63.664,-177.719,7.331,148.717
C07019=1161.323,224.474,-63.688,-177.716,7.333,148.717
C07020=1161.318,224.723,-63.714,-177.713,7.336,148.716
C07021=1161.314,224.971,-63.740,-177.711,7.338,148.716
C07022=1161.309,225.220,-63.765,-177.708,7.340,148.716
C07023=1161.305,225.468,-63.791,-177.705,7.343,148.716
C07024=1161.301,225.717,-63.817,-177.702,7.345,148.716
C07025=1161.296,225.965,-63.842,-177.700,7.348,148.716
C07026=1161.292,226.214,-63.868,-177.697,7.351,148.715
C07027=1161.288,226.463,-63.894,-177.694,7.353,148.715
C07028=1161.283,226.712,-63.920,-177.691,7.356,148.715
C07029=1161.279,226.960,-63.945,-177.689,7.358,148.715
C07030=1161.274,227.209,-63.971,-177.686,7.360,148.715
C07031=1161.269,227.458,-63.997,-177.683,7.363,148.715
C07032=1161.265,227.706,-64.022,-177.681,7.365,148.714
C07033=1161.260,227.955,-64.048,-177.678,7.368,148.714
C07034=1161.256,228.203,-64.074,-177.675,7.371,148.714
C07035=1161.252,228.452,-64.100,-177.673,7.373,148.714
C07036=1161.247,228.700,-64.125,-177.670,7.376,148.714
C07037=1161.243,228.949,-64.151,-177.667,7.379,148.714
C07038=1161.238,229.198,-64.177,-177.665,7.381,148.713
C07039=1161.234,229.446,-64.204,-177.661,7.383,148.713
C07040=1161.229,229.695,-64.229,-177.659,7.386,148.713
C07041=1161.225,229.943,-64.255,-177.656,7.388,148.713
C07042=1161.221,230.192,-64.280,-177.653,7.391,148.713
C07043=1161.216,230.441,-64.307,-177.651,7.393,148.713
C07044=1161.211,230.690,-64.333,-177.648,7.396,148.712
C07045=1161.207,230.938,-64.359,-177.645,7.399,148.712
C07046=1161.203,231.186,-64.384,-177.643,7.401,148.712
C07047=1161.198,231.435,-64.411,-177.640,7.404,148.712
C07048=1161.194,231.684,-64.437,-177.637,7.407,148.712
C07049=1161.190,231.932,-64.463,-177.635,7.409,148.712
C07050=1161.185,232.181,-64.488,-177.632,7.411,148.711
C07051=1161.180,232.430,-64.515,-177.629,7.414,148.711
C07052=1161.176,232.679,-64.540,-177.626,7.417,148.711
C07053=1161.172,232.927,-64.567,-177.624,7.419,148.711
C07054=1161.167,233.176,-64.593,-177.621,7.422,148.711
C07055=1161.162,233.425,-64.619,-177.618,7.425,148.711
C07056=1161.158,233.672,-64.645,-177.615,7.427,148.711
C07057=1161.153,233.921,-64.671,-177.613,7.430,148.710
C07058=1161.149,234.170,-64.697,-177.610,7.433,148.710
C07059=1161.145,234.418,-64.724,-177.607,7.434,148.710
C07060=1161.140,234.667,-64.750,-177.604,7.437,148.710
C07061=1161.136,234.915,-64.777,-177.602,7.440,148.710
C07062=1161.131,235.165,-64.803,-177.599,7.442,148.710
C07063=1161.127,235.413,-64.829,-177.596,7.445,148.709
C07064=1161.122,235.685,-64.857,-177.593,7.448,148.709
C07065=1161.117,235.956,-64.887,-177.590,7.451,148.709
C07066=1161.113,236.228,-64.915,-177.587,7.454,148.709
C07067=1161.107,236.500,-64.944,-177.585,7.457,148.709
C07068=1161.103,236.749,-64.970,-177.581,7.459,148.709
C07069=1161.098,236.996,-64.997,-177.579,7.462,148.709
C07070=1161.094,237.245,-65.022,-177.576,7.464,148.708
C07071=1161.089,237.494,-65.049,-177.574,7.467,148.708
C07072=1161.085,237.742,-65.075,-177.570,7.470,148.708
C07073=1161.080,237.991,-65.102,-177.568,7.472,148.708
C07074=1161.076,238.239,-65.129,-177.565,7.475,148.708
C07075=1161.071,238.488,-65.155,-177.563,7.478,148.708
C07076=1161.067,238.736,-65.181,-177.560,7.481,148.708
C07077=1161.062,238.986,-65.208,-177.557,7.482,148.707
C07078=1161.059,239.234,-65.234,-177.554,7.485,148.707
C07079=1161.054,239.482,-65.261,-177.552,7.488,148.707
C07080=1161.050,239.731,-65.287,-177.549,7.491,148.707
C07081=1161.045,239.980,-65.314,-177.546,7.493,148.707
C07082=1161.041,240.228,-65.341,-177.544,7.496,148.707
C07083=1161.036,240.477,-65.367,-177.541,7.499,148.707
C07084=1161.032,240.725,-65.393,-177.539,7.501,148.707
C07085=1161.028,240.974,-65.420,-177.536,7.504,148.707
C07086=1161.023,241.222,-65.448,-177.533,7.507,148.706
C07087=1161.019,241.471,-65.473,-177.530,7.510,148.706
C07088=1161.014,241.719,-65.500,-177.528,7.512,148.706
C07089=1161.010,241.968,-65.527,-177.525,7.515,148.706
C07090=1161.005,242.216,-65.554,-177.522,7.518,148.706
C07091=1161.000,242.465,-65.580,-177.519,7.520,148.706
C07092=1160.997,242.713,-65.607,-177.517,7.522,148.706
C07093=1160.992,242.962,-65.634,-177.514,7.525,148.706
C07094=1160.987,243.210,-65.661,-177.511,7.528,148.705
C07095=1160.983,243.458,-65.687,-177.508,7.531,148.705
C07096=1160.979,243.707,-65.714,-177.506,7.533,148.705
C07097=1160.974,243.955,-65.741,-177.503,7.536,148.705
C07098=1160.970,244.204,-65.767,-177.500,7.539,148.705
C07099=1160.966,244.454,-65.795,-177.497,7.542,148.705
C07100=1160.961,244.702,-65.822,-177.495,7.544,148.705
C07101=1160.957,244.950,-65.848,-177.492,7.547,148.705
C07102=1160.952,245.199,-65.875,-177.489,7.550,148.704
C07103=1160.948,245.447,-65.902,-177.486,7.552,148.704
C07104=1160.943,245.696,-65.929,-177.484,7.555,148.704
C07105=1160.939,245.944,-65.956,-177.481,7.558,148.704
C07106=1160.935,246.192,-65.983,-177.479,7.560,148.704
C07107=1160.930,246.441,-66.010,-177.476,7.563,148.704
C07108=1160.925,246.689,-66.037,-177.473,7.566,148.704
C07109=1160.921,246.939,-66.064,-177.470,7.568,148.704
C07110=1160.917,247.187,-66.091,-177.468,7.571,148.704
C07111=1160.913,247.435,-66.118,-177.465,7.574,148.703
C07112=1160.908,247.684,-66.145,-177.462,7.577,148.703
C07113=1160.903,247.932,-66.172,-177.459,7.580,148.703
C07114=1160.899,248.181,-66.199,-177.457,7.582,148.703
C07115=1160.895,248.428,-66.226,-177.454,7.585,148.703
C07116=1160.891,248.677,-66.254,-177.451,7.588,148.703
C07117=1160.886,248.926,-66.281,-177.448,7.591,148.703
C07118=1160.882,249.174,-66.308,-177.446,7.593,148.703
C07119=1160.877,249.423,-66.335,-177.443,7.596,148.703
C07120=1160.872,249.671,-66.362,-177.441,7.599,148.703
C07121=1160.869,249.920,-66.390,-177.438,7.602,148.703
C07122=1160.864,250.169,-66.417,-177.435,7.604,148.702
C07123=1160.860,250.417,-66.444,-177.433,7.607,148.702
C07124=1160.855,250.665,-66.471,-177.430,7.609,148.702
C07125=1160.851,250.914,-66.498,-177.427,7.612,148.702
C07126=1160.847,251.162,-66.526,-177.424,7.615,148.702
C07127=1160.842,251.411,-66.553,-177.421,7.618,148.702
C07128=1160.838,251.659,-66.580,-177.419,7.620,148.702
C07129=1160.833,251.907,-66.608,-177.417,7.623,148.702
C07130=1160.829,252.156,-66.635,-177.414,7.626,148.702
C07131=1160.825,252.405,-66.662,-177.411,7.629,148.702
C07132=1160.820,252.653,-66.689,-177.408,7.632,148.702
C07133=1160.816,252.901,-66.717,-177.405,7.635,148.701
C07134=1160.812,253.150,-66.745,-177.403,7.637,148.701
C07135=1160.807,253.398,-66.772,-177.400,7.640,148.701
C07136=1160.803,253.647,-66.799,-177.397,7.643,148.701
C07137=1160.798,253.895,-66.826,-177.394,7.646,148.701
C07138=1160.794,254.144,-66.855,-177.392,7.649,148.701
C07139=1160.789,254.392,-66.882,-177.389,7.651,148.701
C07140=1160.785,254.640,-66.909,-177.387,7.654,148.701
C07141=1160.781,254.889,-66.937,-177.384,7.657,148.701
C07142=1160.777,255.137,-66.965,-177.381,7.659,148.701
C07143=1160.772,255.386,-66.992,-177.378,7.662,148.701
C07144=1160.768,255.634,-67.019,-177.376,7.665,148.700
C07145=1160.764,255.883,-67.047,-177.373,7.668,148.700
C07146=1160.759,256.131,-67.075,-177.371,7.670,148.700
C07147=1160.754,256.380,-67.102,-177.368,7.673,148.700
C07148=1160.750,256.628,-67.130,-177.365,7.676,148.700
C07149=1160.746,256.877,-67.158,-177.362,7.679,148.700
C07150=1160.741,257.124,-67.185,-177.360,7.682,148.700
C07151=1160.737,257.374,-67.213,-177.357,7.685,148.700
C07152=1160.733,257.622,-67.241,-177.355,7.687,148.700
C07153=1160.728,257.870,-67.269,-177.352,7.690,148.700
C07154=1160.724,258.119,-67.296,-177.349,7.693,148.700
C07155=1160.719,258.367,-67.324,-177.346,7.696,148.700
C07156=1160.715,258.616,-67.352,-177.344,7.699,148.700
C07157=1160.711,258.864,-67.379,-177.340,7.702,148.699
C07158=1160.707,259.112,-67.407,-177.338,7.705,148.699
C07159=1160.702,259.361,-67.435,-177.336,7.707,148.699
C07160=1160.697,259.609,-67.463,-177.333,7.710,148.699
C07161=1160.694,259.858,-67.491,-177.330,7.713,148.699
C07162=1160.689,260.106,-67.519,-177.327,7.716,148.699
C07163=1160.684,260.354,-67.546,-177.324,7.719,148.699
C07164=1160.680,260.603,-67.575,-177.322,7.722,148.699
C07165=1160.676,260.851,-67.602,-177.319,7.725,148.699
C07166=1160.672,261.099,-67.630,-177.317,7.727,148.699
C07167=1160.667,261.348,-67.658,-177.314,7.730,148.699
C07168=1160.662,261.621,-67.690,-177.311,7.733,148.699
C07169=1160.658,261.894,-67.720,-177.308,7.736,148.699
C07170=1160.653,262.168,-67.751,-177.305,7.739,148.699
C07171=1160.648,262.441,-67.782,-177.302,7.742,148.699
C07172=1160.644,262.689,-67.809,-177.300,7.745,148.698
C07173=1160.639,262.938,-67.838,-177.297,7.748,148.698
C07174=1160.635,263.186,-67.866,-177.294,7.751,148.698
C07175=1160.631,263.435,-67.893,-177.291,7.754,148.698
C07176=1160.626,263.683,-67.922,-177.289,7.757,148.698
C07177=1160.622,263.932,-67.950,-177.286,7.760,148.698
C07178=1160.617,264.180,-67.978,-177.283,7.763,148.698
C07179=1160.613,264.428,-68.006,-177.281,7.765,148.698
C07180=1160.609,264.676,-68.034,-177.279,7.768,148.698
C07181=1160.605,264.925,-68.063,-177.276,7.771,148.698
C07182=1160.600,265.173,-68.091,-177.273,7.774,148.698
C07183=1160.596,265.422,-68.119,-177.270,7.777,148.698
C07184=1160.591,265.670,-68.147,-177.267,7.780,148.698
C07185=1160.587,265.919,-68.176,-177.265,7.783,148.698
C07186=1160.582,266.166,-68.204,-177.262,7.786,148.698
C07187=1160.579,266.415,-68.232,-177.259,7.789,148.698
C07188=1160.574,266.663,-68.260,-177.256,7.792,148.698
C07189=1160.570,266.911,-68.289,-177.254,7.794,148.698
C07190=1160.565,267.159,-68.317,-177.251,7.797,148.698
C07191=1160.561,267.408,-68.346,-177.249,7.800,148.698
C07192=1160.556,267.656,-68.374,-177.246,7.803,148.698
C07193=1160.553,267.905,-68.402,-177.243,7.806,148.697
C07194=1160.548,268.154,-68.431,-177.241,7.809,148.698
C07195=1160.544,268.401,-68.459,-177.238,7.812,148.698
C07196=1160.539,268.650,-68.487,-177.235,7.815,148.698
C07197=1160.534,268.898,-68.516,-177.233,7.818,148.697
C07198=1160.531,269.147,-68.545,-177.230,7.821,148.697
C07199=1160.526,269.395,-68.573,-177.227,7.824,148.697
C07200=1160.522,269.643,-68.601,-177.224,7.827,148.697
C07201=1160.518,269.892,-68.631,-177.222,7.829,148.697
C07202=1160.513,270.139,-68.658,-177.219,7.832,148.697
C07203=1160.509,270.388,-68.687,-177.217,7.835,148.697
C07204=1160.504,270.637,-68.716,-177.214,7.838,148.697
C07205=1160.500,270.884,-68.744,-177.212,7.841,148.697
C07206=1160.496,271.133,-68.773,-177.209,7.844,148.697
C07207=1160.492,271.382,-68.801,-177.206,7.847,148.697
C07208=1160.487,271.629,-68.830,-177.203,7.850,148.697
C07209=1160.483,271.878,-68.859,-177.200,7.853,148.697
C07210=1160.479,272.127,-68.887,-177.198,7.856,148.697
C07211=1160.474,272.374,-68.916,-177.195,7.859,148.697
C07212=1160.470,272.623,-68.945,-177.193,7.862,148.697
C07213=1160.466,272.871,-68.974,-177.190,7.865,148.697
C07214=1160.461,273.120,-69.002,-177.187,7.868,148.697
C07215=1160.457,273.368,-69.032,-177.184,7.871,148.697
C07216=1160.453,273.616,-69.060,-177.182,7.873,148.697
C07217=1160.448,273.865,-69.088,-177.179,7.876,148.697
C07218=1160.444,274.113,-69.118,-177.177,7.879,148.697
C07219=1160.440,274.362,-69.146,-177.174,7.882,148.697
C07220=1160.436,274.610,-69.175,-177.172,7.885,148.697
C07221=1160.431,274.858,-69.204,-177.169,7.888,148.697
C07222=1160.427,275.106,-69.233,-177.166,7.891,148.697
C07223=1160.423,275.354,-69.262,-177.163,7.894,148.697
C07224=1160.418,275.602,-69.290,-177.161,7.897,148.697
C07225=1160.414,275.851,-69.320,-177.158,7.900,148.697
C07226=1160.410,276.099,-69.348,-177.156,7.903,148.697
C07227=1160.405,276.348,-69.378,-177.153,7.906,148.697
C07228=1160.401,276.597,-69.407,-177.150,7.909,148.697
C07229=1160.397,276.844,-69.435,-177.147,7.912,148.697
C07230=1160.393,277.092,-69.465,-177.145,7.915,148.697
C07231=1160.388,277.341,-69.493,-177.142,7.918,148.697
C07232=1160.384,277.589,-69.523,-177.139,7.921,148.697
C07233=1160.379,277.837,-69.552,-177.137,7.924,148.697
C07234=1160.375,278.086,-69.581,-177.134,7.927,148.697
C07235=1160.371,278.334,-69.609,-177.132,7.931,148.697
C07236=1160.367,278.582,-69.639,-177.129,7.934,148.697
C07237=1160.363,278.830,-69.668,-177.126,7.937,148.697
C07238=1160.358,279.078,-69.697,-177.123,7.939,148.697
C07239=1160.354,279.327,-69.726,-177.121,7.943,148.697
C07240=1160.350,279.575,-69.756,-177.118,7.946,148.697
C07241=1160.345,279.823,-69.785,-177.115,7.949,148.697
C07242=1160.341,280.072,-69.814,-177.113,7.952,148.697
C07243=1160.337,280.320,-69.843,-177.110,7.955,148.697
C07244=1160.332,280.568,-69.872,-177.108,7.958,148.697
C07245=1160.328,280.816,-69.902,-177.105,7.961,148.697
C07246=1160.324,281.064,-69.931,-177.102,7.964,148.697
C07247=1160.320,281.312,-69.960,-177.099,7.967,148.697
C07248=1160.316,281.561,-69.990,-177.097,7.970,148.697
C07249=1160.311,281.810,-70.018,-177.094,7.973,148.697
C07250=1160.307,282.058,-70.048,-177.092,7.976,148.697
C07251=1160.302,282.305,-70.077,-177.089,7.979,148.697
C07252=1160.298,282.554,-70.107,-177.087,7.982,148.697
C07253=1160.293,282.802,-70.136,-177.084,7.985,148.697
C07254=1160.289,283.051,-70.166,-177.081,7.988,148.697
C07255=1160.285,283.299,-70.195,-177.078,7.991,148.697
C07256=1160.281,283.547,-70.225,-177.076,7.994,148.697
C07257=1160.277,283.795,-70.254,-177.073,7.997,148.697
C07258=1160.272,284.044,-70.284,-177.070,8.000,148.697
C07259=1160.268,284.292,-70.313,-177.068,8.003,148.697
C07260=1160.264,284.540,-70.343,-177.065,8.006,148.697
C07261=1160.260,284.788,-70.372,-177.063,8.009,148.697
C07262=1160.255,285.036,-70.401,-177.060,8.012,148.697
C07263=1160.251,285.284,-70.431,-177.058,8.016,148.697
C07264=1160.247,285.532,-70.460,-177.055,8.019,148.697
C07265=1160.242,285.780,-70.491,-177.052,8.022,148.697
C07266=1160.238,286.029,-70.520,-177.049,8.025,148.697
C07267=1160.234,286.277,-70.550,-177.047,8.028,148.697
C07268=1160.230,286.525,-70.579,-177.044,8.031,148.697
C07269=1160.225,286.774,-70.609,-177.041,8.034,148.697
C07270=1160.221,287.022,-70.638,-177.039,8.037,148.697
C07271=1160.216,287.270,-70.668,-177.036,8.040,148.697
C07272=1160.212,287.545,-70.701,-177.034,8.043,148.697
C07273=1160.207,287.820,-70.733,-177.031,8.047,148.697
C07274=1160.203,288.095,-70.767,-177.028,8.050,148.697
C07275=1160.198,288.370,-70.800,-177.025,8.054,148.697
C07276=1160.193,288.618,-70.830,-177.022,8.057,148.697
C07277=1160.189,288.867,-70.860,-177.020,8.060,148.697
C07278=1160.185,289.115,-70.889,-177.017,8.063,148.697
C07279=1160.181,289.362,-70.919,-177.014,8.066,148.697
C07280=1160.176,289.611,-70.949,-177.012,8.069,148.698
C07281=1160.172,289.859,-70.979,-177.009,8.072,148.698
C07282=1160.168,290.107,-71.009,-177.006,8.075,148.698
C07283=1160.164,290.356,-71.039,-177.004,8.078,148.698
C07284=1160.160,290.605,-71.069,-177.001,8.081,148.698
C07285=1160.156,290.852,-71.099,-176.998,8.084,148.698
C07286=1160.152,291.100,-71.128,-176.996,8.088,148.698
C07287=1160.147,291.348,-71.159,-176.993,8.091,148.698
C07288=1160.143,291.597,-71.189,-176.991,8.094,148.698
C07289=1160.139,291.845,-71.218,-176.988,8.097,148.698
C07290=1160.134,292.093,-71.249,-176.986,8.100,148.698
C07291=1160.130,292.341,-71.278,-176.983,8.103,148.698
C07292=1160.126,292.589,-71.308,-176.981,8.106,148.698
C07293=1160.121,292.837,-71.338,-176.978,8.109,148.698
C07294=1160.117,293.085,-71.369,-176.975,8.113,148.698
C07295=1160.113,293.334,-71.398,-176.972,8.116,148.698
C07296=1160.109,293.582,-71.429,-176.969,8.119,148.698
C07297=1160.105,293.830,-71.459,-176.967,8.122,148.698
C07298=1160.100,294.078,-71.489,-176.964,8.125,148.698
C07299=1160.096,294.326,-71.520,-176.962,8.129,148.698
C07300=1160.091,294.574,-71.550,-176.959,8.131,148.698
C07301=1160.087,294.822,-71.580,-176.957,8.134,148.698
C07302=1160.084,295.071,-71.610,-176.954,8.138,148.699
C07303=1160.079,295.319,-71.640,-176.951,8.141,148.699
C07304=1160.075,295.567,-71.671,-176.949,8.144,148.699
C07305=1160.070,295.815,-71.701,-176.946,8.147,148.699
C07306=1160.067,296.063,-71.731,-176.944,8.150,148.699
C07307=1160.062,296.311,-71.761,-176.941,8.153,148.699
C07308=1160.058,296.560,-71.791,-176.939,8.156,148.699
C07309=1160.054,296.808,-71.822,-176.936,8.160,148.699
C07310=1160.050,297.055,-71.852,-176.933,8.163,148.699
C07311=1160.045,297.303,-71.883,-176.931,8.166,148.699
C07312=1160.041,297.552,-71.912,-176.928,8.169,148.699
C07313=1160.037,297.800,-71.944,-176.925,8.172,148.699
C07314=1160.033,298.048,-71.974,-176.923,8.176,148.699
C07315=1160.029,298.296,-72.005,-176.920,8.179,148.699
C07316=1160.024,298.544,-72.035,-176.918,8.182,148.699
C07317=1160.020,298.793,-72.065,-176.915,8.185,148.699
C07318=1160.016,299.041,-72.096,-176.913,8.188,148.700
C07319=1160.012,299.288,-72.126,-176.910,8.191,148.700
C07320=1160.007,299.536,-72.157,-176.907,8.195,148.700
C07321=1160.003,299.785,-72.188,-176.904,8.198,148.700
C07322=1159.999,300.033,-72.218,-176.902,8.201,148.700
C07323=1159.995,300.281,-72.249,-176.899,8.204,148.700
C07324=1159.990,300.529,-72.280,-176.897,8.207,148.700
C07325=1159.987,300.778,-72.309,-176.894,8.211,148.700
C07326=1159.982,301.026,-72.340,-176.891,8.214,148.700
C07327=1159.977,301.273,-72.371,-176.889,8.217,148.700
C07328=1159.973,301.521,-72.401,-176.886,8.220,148.700
C07329=1159.969,301.770,-72.432,-176.884,8.223,148.700
C07330=1159.965,302.018,-72.463,-176.881,8.227,148.700
